# B&R Automation Studio project PLC code - cp (part 8)

#### Status.st
```iecst
ACTION Status:

	CASE Primer.Status.DeviceStatus OF
		PRIMER_TURNED_OFF:
			IF Primer.Inputs.xPrimerPresent THEN
				Primer.Status.DeviceStatus:=PRIMER_INIT;
			END_IF

		PRIMER_INIT:
			IF NOT Primer.Inputs.xPrimerPresent THEN
				Primer.Status.DeviceStatus:=PRIMER_TURNED_OFF;
			ELSIF Primer.Outputs.Physical.xPrepareToPrime OR Primer.Outputs.Physical.xRunTransport THEN
				Primer.Status.DeviceStatus:=PRIMER_PREPARING;
			END_IF

		PRIMER_PREPARING:
			IF Primer.Inputs.xTransportMoving THEN
				Primer.Status.DeviceStatus:=PRIMER_BELT_RUNNING;
			ELSIF NOT Primer.Outputs.Physical.xPrepareToPrime AND NOT Primer.Outputs.Physical.xRunTransport THEN
				Primer.Status.DeviceStatus:=PRIMER_INIT;
			END_IF

		PRIMER_BELT_RUNNING:
			IF NOT Primer.Inputs.xTransportMoving THEN
				Primer.Status.DeviceStatus:=PRIMER_INIT;
			END_IF
			IF Primer.Inputs.xReadyToPrime THEN
				Primer.Status.DeviceStatus:=PRIMER_READY;
			END_IF

		PRIMER_READY:
			IF NOT Primer.Inputs.xReadyToPrime THEN
				Primer.Status.DeviceStatus:=PRIMER_BELT_RUNNING;
			END_IF
			IF Primer.Inputs.xCoating THEN
				Primer.Status.DeviceStatus:=PRIMER_PRIMING;
			END_IF

		PRIMER_PRIMING:
			IF NOT Primer.Inputs.xCoating THEN
				Primer.Status.DeviceStatus:=PRIMER_READY;
			END_IF
			IF Primer.Inputs.xDryerInRun THEN
				Primer.Status.DeviceStatus:=PRIMER_DRYING;
			END_IF

		PRIMER_DRYING:
			IF NOT Primer.Inputs.xDryerInRun THEN
				Primer.Status.DeviceStatus:=PRIMER_PRIMING;
			END_IF

		PRIMER_FAULTED:
			IF NOT Primer.Inputs.xError THEN
				Primer.Status.DeviceStatus:=PRIMER_TURNED_OFF;
			END_IF

	END_CASE

	IF NOT Primer.Inputs.xPrimerPresent THEN
		Primer.Status.DeviceStatus:=PRIMER_TURNED_OFF;
	END_IF
	IF Primer.Status.DeviceStatus <> PRIMER_TURNED_OFF AND Primer.Inputs.xError THEN
		Primer.Status.DeviceStatus:=PRIMER_FAULTED;
	END_IF

	UpdateStatus;

	//Empty belt status
	tiTimeToEmpty := REAL_TO_TIME(60 * (Primer.Parameters.Hw.rPrimerLength + Primer.Parameters.rMediaLength) / Primer.Parameters.rSpeedSetPoint);
	tonEmptyBelt.IN := Primer.Inputs.xTransportMoving;
	tonEmptyBelt.PT := tiTimeToEmpty;
	tonEmptyBelt();
	IF Primer.Status.Comms.xModuleOk THEN
		Primer.Status.xBeltEmpty := Primer.Inputs.Comms.xBeltEmpty AND (tonEmptyBelt.Q OR NOT Primer.Inputs.xTransportMoving);
	ELSE
		Primer.Status.xBeltEmpty := (tonEmptyBelt.Q OR NOT Primer.Inputs.xTransportMoving);
	END_IF

END_ACTION

ACTION UpdateStatus:

	Primer.Status.Device.xTurnedOff 	:=	Primer.Status.DeviceStatus=PRIMER_TURNED_OFF;
	Primer.Status.Device.xInit			:=	Primer.Status.DeviceStatus=PRIMER_INIT;
	Primer.Status.Device.xPreparing 	:=	Primer.Status.DeviceStatus=PRIMER_PREPARING;
	Primer.Status.Device.xReady			:=	Primer.Status.DeviceStatus=PRIMER_READY;
	Primer.Status.Device.xPriming 		:=	Primer.Status.DeviceStatus=PRIMER_PRIMING;
	Primer.Status.Device.xFaulted 		:=	Primer.Status.DeviceStatus=PRIMER_FAULTED;

END_ACTION
```

### PrimerSim.typ
```iecst
TYPE
	PrimerSimCommands_typ : 	STRUCT
		CreateError : BOOL;
	END_STRUCT;
	PrimerSim_typ : 	STRUCT
		Commands : PrimerSimCommands_typ;
	END_STRUCT;
END_TYPE
```

### Program Logical/ExtPack/_Ancillaries/PrimerCtrl/PrimerSim/PrimerSim_v1/PrimerSim (IEC)

#### PrimerSim.st - Init, cyclic, exit code
```iecst
PROGRAM _INIT

	Primer ACCESS ADR(gPrimer);
	SimPrimer ACCESS ADR(gSimPrimer);

	Primer.Status.Comms.xModuleOk := TRUE;

END_PROGRAM

PROGRAM _CYCLIC
	(* Insert code here *)
	Primer ACCESS ADR(gPrimer);
	SimPrimer ACCESS ADR(gSimPrimer);

	IF NOT Primer.Parameters.xInstalled THEN
		Primer.Inputs := PrimerInputsReseted;
		RETURN;
	END_IF

	Primer.Inputs.xPrimerPresent:=TRUE;
	Primer.Inputs.Comms.xRemote := TRUE;
	Primer.Inputs.xError:=SimPrimer.Commands.CreateError;

	tonTransport.IN:= Primer.Outputs.Physical.xRunTransport;
	tonTransport.PT:= T#1s;
	tonTransport();
	Primer.Inputs.xTransportMoving:=tonTransport.Q;

	tonReady.IN:= Primer.Inputs.xTransportMoving AND Primer.Outputs.Physical.xPrepareToPrime;
	tonReady.PT:= T#2s;
	tonReady();
	Primer.Inputs.xReadyToPrime:=tonReady.Q;

	tonPrime.IN:= Primer.Inputs.xReadyToPrime AND Primer.Outputs.Physical.xRunPriming;
	tonPrime.PT:= T#1s;
	tonPrime();
	Primer.Inputs.xCoating:=tonPrime.Q;

	tonDry.IN:= Primer.Inputs.xCoating AND Primer.Outputs.Physical.xRunDryer;
	tonDry.PT:= T#1s;
	tonDry();
	Primer.Inputs.xDryerInRun:=tonDry.Q;

	Primer.Inputs.Comms.xBeltEmpty:=TRUE;
	Primer.Inputs.Comms.xCommsOK:=TRUE;

END_PROGRAM
```

#### PrimerSim.var - Local variables
```iecst
VAR
	SimPrimer : REFERENCE TO PrimerSim_typ;
	Primer : REFERENCE TO Primer_typ;
	tonTransport : TON;
	tonReady : TON;
	tonPrime : TON;
	tonBeltEmpty : TON;
	tonDry : TON;
	PrimerInputsReseted : {REDUND_UNREPLICABLE} PrimerInputs_typ;
END_VAR
```

- Dryer.graphml (not shown)

### Program Logical/ExtPack/_Ancillaries/DryerCtrl/DryerCtrl_v1/DryerCtrl (IEC)

#### Status.st
```iecst
ACTION Status:

	CASE Dryer.Status.DeviceStatus OF
		DRYER_TURNED_OFF:
			IF Dryer.Inputs.xInRemote THEN
				Dryer.Status.DeviceStatus:=DRYER_INIT;
			END_IF

		DRYER_INIT:
			IF Dryer.Outputs.xRunTransport OR Dryer.Outputs.xPrepareToDry THEN
				Dryer.Status.DeviceStatus:=DRYER_PREPARING;
			END_IF

		DRYER_PREPARING:
			IF Dryer.Inputs.xTransportMoving THEN
				Dryer.Status.DeviceStatus:=DRYER_BELTRUNNING;
			ELSIF NOT Dryer.Outputs.xRunTransport AND NOT Dryer.Outputs.xPrepareToDry THEN
				Dryer.Status.DeviceStatus:=DRYER_INIT;
			END_IF

		DRYER_BELTRUNNING:
			IF Dryer.Inputs.xReadyToDry THEN
				Dryer.Status.DeviceStatus:=DRYER_READY;
			ELSIF NOT Dryer.Inputs.xTransportMoving THEN
				Dryer.Status.DeviceStatus:=DRYER_INIT;
			END_IF

		DRYER_READY:
			IF Dryer.Inputs.xDrying THEN
				Dryer.Status.DeviceStatus:=DRYER_DRYING;
			ELSIF NOT Dryer.Inputs.xReadyToDry THEN
				Dryer.Status.DeviceStatus:=DRYER_INIT;
			END_IF

		DRYER_DRYING:
			IF NOT Dryer.Inputs.xDrying THEN
				Dryer.Status.DeviceStatus:=DRYER_INIT;
			END_IF

		DRYER_FAULTED:
			IF NOT Dryer.Inputs.xError THEN
				Dryer.Status.DeviceStatus:=DRYER_INIT;
			END_IF

	END_CASE

	IF NOT Dryer.Inputs.xCommsOK THEN
		Dryer.Status.DeviceStatus:=DRYER_TURNED_OFF;
	END_IF
	IF Dryer.Status.DeviceStatus <> DRYER_TURNED_OFF AND Dryer.Inputs.xError THEN
		Dryer.Status.DeviceStatus:=DRYER_FAULTED;
	END_IF

	UpdateStatus;

	//Empty belt status
	tiTimeToEmpty := REAL_TO_TIME(60 * (Dryer.Parameters.Hw.rDryerLength + Dryer.Parameters.rMediaLength) / Dryer.Parameters.rSpeedSetPoint);
	tonEmptyBelt.IN := Dryer.Inputs.xTransportMoving;
	tonEmptyBelt.PT := tiTimeToEmpty;
	tonEmptyBelt();
	IF Dryer.Inputs.xCommsOK THEN
		Dryer.Status.xBeltEmpty := Dryer.Inputs.xBeltEmpty AND (tonEmptyBelt.Q OR NOT Dryer.Inputs.xTransportMoving);
	ELSE
		Dryer.Status.xBeltEmpty := (tonEmptyBelt.Q OR NOT Dryer.Inputs.xTransportMoving);
	END_IF

END_ACTION

ACTION UpdateStatus:

	Dryer.Status.Device.xTurnedOff 		:=	Dryer.Status.DeviceStatus=DRYER_TURNED_OFF;
	Dryer.Status.Device.xInit 			:=	Dryer.Status.DeviceStatus=DRYER_INIT;
	Dryer.Status.Device.xPreparing 		:=	Dryer.Status.DeviceStatus=DRYER_PREPARING;
	Dryer.Status.Device.xBeltRunning 	:=	Dryer.Status.DeviceStatus=DRYER_BELTRUNNING;
	Dryer.Status.Device.xReadyToDry 	:=	Dryer.Status.DeviceStatus=DRYER_READY;
	Dryer.Status.Device.xDrying 		:=	Dryer.Status.DeviceStatus=DRYER_DRYING;
	Dryer.Status.Device.xFaulted 		:=	Dryer.Status.DeviceStatus=DRYER_FAULTED;

END_ACTION
```

#### Alarms.st
```iecst
ACTION Alarms:

	Dryer.Alarms.xNoDryerPresent:= NOT Dryer.Inputs.xInRemote;

	//IF NO Dryer, define that alarm and exit
	IF Dryer.Alarms.xNoDryerPresent THEN
		ResetAlarms;
		Dryer.Alarms.xNoDryerPresent:=TRUE;
	END_IF

	//Error
	IF Dryer.Inputs.xError THEN
		Dryer.Alarms.xError := TRUE;
	END_IF

	//Remote
	IF (NOT Dryer.Inputs.xInRemote) AND Dryer.Parameters.xLineInAuto THEN
		Dryer.Alarms.xNotRemote := TRUE;
	END_IF

	//Stop request
	IF (Dryer.Inputs.xStopButtonPressed) THEN
		Dryer.Alarms.xStopRequest := TRUE;
	END_IF

	//Summary
	Dryer.Alarms.xCriticalAlarm:= 	Dryer.Alarms.xError OR
									Dryer.Alarms.xNotRemote OR
									Dryer.Alarms.xStopRequest;

END_ACTION

ACTION ResetAlarms:
	Dryer.Alarms := AlarmsReseted;
END_ACTION
```

### Program Logical/ExtPack/_Ancillaries/OpvCtrl/OpvCtrl_v1/OpvCtrl (IEC)

#### Opv.st - Init, cyclic, exit code
```iecst
PROGRAM _CYCLIC

	OverVarnish ACCESS ADR(gOverVarnish);

	//Version
	OverVarnish.Status.Version.iVersion0 := OverVarnish.Inputs.Comms.iVersion1;
	OverVarnish.Status.Version.iVersion1 := OverVarnish.Inputs.Comms.iVersion2;
	OverVarnish.Status.Version.iVersion2 := OverVarnish.Inputs.Comms.iVersion3;
	OverVarnish.Status.Version.iVersion3 := OverVarnish.Inputs.Comms.iVersion4;

	//Model evaluation
	iOpvModel.0 := OverVarnish.Inputs.xModelInput[0];
	iOpvModel.1 := OverVarnish.Inputs.xModelInput[1];
	iOpvModel.2 := OverVarnish.Inputs.xModelInput[2];

	OverVarnish.Parameters.xInstalled := iOpvModel>0;

	//Specify Type of Opv Model
	OverVarnish.Status.iModel := iOpvModel;
	CASE iOpvModel OF
		1: OverVarnish.Status.OpvType := OPVTY_GIARDINA;
		2: OverVarnish.Status.OpvType := OPVTY_DMS;
		3: OverVarnish.Status.OpvType := OPVTY_TECLIGHTING;
		ELSE OverVarnish.Status.OpvType := OPVTY_UNDEFINED;
	END_CASE

	IF NOT OverVarnish.Parameters.xInstalled OR NOT OverVarnish.ParSw.xEnabled THEN
		ResetAlarms;
		OverVarnish.Outputs := OutputsReset;
		OverVarnish.Commands:=ResetCommands;
		OverVarnish.Status.DeviceStatus:=OPV_TURNED_OFF;
		CopyOfWriteData := EraseWriteData;
		UpdateStatus;
		RETURN;
	END_IF

	IF OverVarnish.Commands.xResetAlarms THEN ResetAlarms; END_IF

	Configuration;

	IF NOT OverVarnish.Parameters.xSimulationMode THEN
		AssignDataComms;
	END_IF

	Status;

	//Erasing data when ancillary not in remote
	IF NOT OverVarnish.Inputs.Comms.xRemote THEN
		CopyOfWriteData := EraseWriteData;
	END_IF

	Alarms;

	IF OverVarnish.Status.Device.xFaulted OR OverVarnish.Status.Device.xTurnedOff OR NOT OverVarnish.Parameters.xLineInAuto THEN
		OverVarnish.Status.CtrlStatus:=OPVCTRL_STOPPED;
	END_IF

	CASE OverVarnish.Status.CtrlStatus OF
		OPVCTRL_STOPPED:
			//Actions
			OverVarnish.Outputs.Physical := PhysicalOutputsReset;

			//Transition
			IF OverVarnish.Commands.xPrepare THEN
				xEnablePriming:= OverVarnish.ParSw.xEnablePriming AND OverVarnish.Orders.xEnablePriming;
				OverVarnish.Status.CtrlStatus:=OPVCTRL_PREPARING;
			END_IF

		OPVCTRL_STOPPING:
			//Actions
			OverVarnish.Outputs.Physical := PhysicalOutputsReset;

			//Transition
			IF OverVarnish.Status.DeviceStatus=OPV_TURNED_OFF OR OverVarnish.Status.DeviceStatus=OPV_INIT THEN
				OverVarnish.Status.CtrlStatus:=OPVCTRL_STOPPED;
			END_IF

		OPVCTRL_CONTROLSTOPPING:
			//Wait to have the belt empty and send the Stop order
			IF OverVarnish.Status.xBeltEmpty AND EDGEPOS(OverVarnish.Orders.xDisableReadBlock) OR NOT OverVarnish.Inputs.xTransportMoving THEN
				OverVarnish.Status.CtrlStatus:=OPVCTRL_STOPPING;
			END_IF

		OPVCTRL_PREPARING:
			//Actions

			IF xEnablePriming THEN
				OverVarnish.Outputs.Physical.xRunTransport:=TRUE;
				OverVarnish.Outputs.Physical.xPrepareToPrime:=TRUE;
				//Transition
				IF OverVarnish.Status.DeviceStatus=OPV_READY THEN
					OverVarnish.Status.CtrlStatus:=OPVCTRL_PREPARED;
				END_IF

			ELSE
				OverVarnish.Outputs.Physical.xRunTransport:=TRUE;
				//Transition
				IF OverVarnish.Status.DeviceStatus=OPV_BELT_RUNNING THEN
					OverVarnish.Status.CtrlStatus:=OPVCTRL_PREPARED;
				END_IF

			END_IF

		OPVCTRL_PAUSED,
		OPVCTRL_PREPARED:
			//Actions
			IF OverVarnish.Commands.xStart THEN
				OverVarnish.Status.CtrlStatus:=OPVCTRL_STARTING;
			END_IF

		OPVCTRL_STARTING:
			//Actions
			IF xEnablePriming THEN
				OverVarnish.Outputs.Physical.xRunPriming:=TRUE;
				IF OverVarnish.Status.DeviceStatus=OPV_PRIMING THEN
					OverVarnish.Outputs.Physical.xRunDryer:=TRUE;
				END_IF
				//Transition
				IF OverVarnish.Status.DeviceStatus=OPV_DRYING THEN
					OverVarnish.Status.CtrlStatus:=OPVCTRL_WORKING;
				END_IF

			ELSE
				OverVarnish.Outputs.Physical.xRunTransport:=TRUE;
				IF OverVarnish.Status.DeviceStatus=OPV_BELT_RUNNING THEN
					OverVarnish.Status.CtrlStatus:=OPVCTRL_WORKING;
				END_IF

			END_IF

			//Transition
			IF OverVarnish.Commands.xPause THEN
				OverVarnish.Status.CtrlStatus:=OPVCTRL_PAUSING;
			END_IF

		OPVCTRL_WORKING:
			IF OverVarnish.Commands.xPause THEN
				OverVarnish.Status.CtrlStatus:=OPVCTRL_PAUSING;
			END_IF

		OPVCTRL_PAUSING:
			//Wait to empty the Belt to avoid media inside
			IF OverVarnish.Status.xBeltEmpty THEN
				IF xEnablePriming THEN
					OverVarnish.Outputs.Physical.xRunDryer:=FALSE;
					//Transition
					IF OverVarnish.Status.DeviceStatus=OPV_PRIMING THEN
						OverVarnish.Status.CtrlStatus:=OPVCTRL_PAUSED;
					END_IF

				ELSE
					IF OverVarnish.Status.DeviceStatus=OPV_INIT OR OverVarnish.Status.DeviceStatus=OPV_BELT_RUNNING THEN
						OverVarnish.Status.CtrlStatus:=OPVCTRL_PAUSED;
					END_IF
				END_IF
			END_IF

	END_CASE

	IF OverVarnish.Commands.xStop THEN
		OverVarnish.Status.CtrlStatus:=OPVCTRL_STOPPING;
	ELSIF OverVarnish.Commands.xControlStop THEN
		OverVarnish.Status.CtrlStatus:=OPVCTRL_CONTROLSTOPPING;
	END_IF

	//Store the history of the status to easy the debug
	IF OverVarnish.Status.CtrlStatus<>StateHistory[0] THEN
		FOR iIndexHistory:=iHistoryLines TO 1 BY -1 DO
			StateHistory[iIndexHistory]:=StateHistory[iIndexHistory-1];
		END_FOR;
		StateHistory[0]:=OverVarnish.Status.CtrlStatus;
	END_IF

	//Fall down the commands
	OverVarnish.Commands:=ResetCommands;

END_PROGRAM
```

#### AssignDataComms.st
```iecst
ACTION AssignDataComms:

	//Active modbus slave diagnosis when ancillary is enabled. This parameter must remain to TRUE from then on.
	//Just would be set to FALSE via UaExpert, to reset historic errors when ancillary is disabled
	OverVarnish.Parameters.xActiveSlaveDiagnosis := TRUE;

	xBoardParametersChanged := 	(OverVarnish.Parameters.Media.rWidth<>rPrevWidth) OR
								(OverVarnish.Parameters.Media.rLength<>rPrevLength) OR
								(OverVarnish.Parameters.Media.rThickness<>rPrevThickness) OR
								(OverVarnish.Parameters.Media.rGap<>rPrevGap);

	rPrevWidth:=OverVarnish.Parameters.Media.rWidth;
	rPrevLength:=OverVarnish.Parameters.Media.rLength;
	rPrevThickness:=OverVarnish.Parameters.Media.rThickness;
	rPrevGap:=OverVarnish.Parameters.Media.rGap;

	tof_BoardParametersChanged.IN:=xBoardParametersChanged;
	tof_BoardParametersChanged.PT:=t#1s;
	tof_BoardParametersChanged();

	IF OverVarnish.Status.OpvType = OPVTY_DMS THEN
		DmsComms;
	ELSE
		DefaultPrimerComms;
	END_IF

	//Disabling writting after some time active. To test
	tonDisableWrittingOfData.IN:= NOT xDisableWriteData;
	tonDisableWrittingOfData.PT:= T#1000ms;
	tonDisableWrittingOfData();

	IF tonDisableWrittingOfData.Q THEN
		xDisableWriteData := TRUE;
	END_IF

	FOR iIndex:=1 TO 25 DO
		IF gToWriteDataModbOpv[iIndex]<>CopyOfWriteData[iIndex] THEN
			xDisableWriteData := FALSE;
		END_IF
	END_FOR

	OverVarnish.Orders.xDisableWriteBlock := xDisableWriteData;

	//Copying previous data
	CopyOfWriteData := gToWriteDataModbOpv;

END_ACTION

ACTION DmsComms:

			/////////////////
			//Pre bits treatment
			OverVarnish.Outputs.Comms.iControl.1 := OverVarnish.Commands.xEnteringMedia;
			OverVarnish.Outputs.Comms.iControl.2 := OverVarnish.Commands.xNewBoardParameters:=tof_BoardParametersChanged.Q;
			//OverVarnish.Outputs.Comms.iControl.3 := ;
			OverVarnish.Outputs.Comms.iControl.4 := TRUE; //OverVarnish.Outputs.Comms.xLineAirSupply;
			OverVarnish.Outputs.Comms.iControl.5 := OverVarnish.Parameters.LineState = LINE_PREPARING_EMPTYBELT OR
													OverVarnish.Parameters.LineState = LINE_STARTING_EMPTYBELT OR
													OverVarnish.Parameters.LineState = LINE_BELT_EMPTYING;

			OverVarnish.Outputs.Comms.iControl2.13 := FALSE; //Single line:0, Double line: 1
			OverVarnish.Outputs.Comms.iControl2.15 := TRUE; //Edge:0, Center: 1

			//Write Registers
			gToWriteDataModbOpv[1] := REAL_TO_UINT(OverVarnish.Parameters.Media.rWidth*10);
			gToWriteDataModbOpv[2] := REAL_TO_UINT(OverVarnish.Parameters.Media.rLength*10);
			gToWriteDataModbOpv[3] := REAL_TO_UINT(OverVarnish.Parameters.Media.rThickness*10);
			gToWriteDataModbOpv[4] := REAL_TO_UINT(OverVarnish.Parameters.Media.rGap*10);
			//gToWriteDataModbOpv[5] := ;
			gToWriteDataModbPrimer[6] := REAL_TO_UINT(OverVarnish.Parameters.rLineAccelRate*60); //150;
			gToWriteDataModbPrimer[7] := REAL_TO_UINT(OverVarnish.Parameters.rLineDecelRate*60); //150;
			gToWriteDataModbOpv[8] := REAL_TO_UINT(OverVarnish.Parameters.rSpeedSetPoint*100);
			gToWriteDataModbOpv[9] := OverVarnish.Outputs.Comms.iControl;
			gToWriteDataModbOpv[10] := OverVarnish.Outputs.Comms.iControl2;
			//gToWriteDataModbOpv[11] := ;
			//gToWriteDataModbOpv[12] := ;
			//gToWriteDataModbOpv[13] := ;
			gToWriteDataModbOpv[14] := REAL_TO_UINT(OverVarnish.Parameters.rLineAccelRate*60); //150;
			gToWriteDataModbOpv[15] := REAL_TO_UINT(OverVarnish.Parameters.rLineDecelRate*60); //150;
			(*
			gToWriteDataModbOpv[16] := ;
			gToWriteDataModbOpv[17] := ;
			gToWriteDataModbOpv[18] := ;
			gToWriteDataModbOpv[19] := ;
			gToWriteDataModbOpv[20] := ;
			gToWriteDataModbOpv[21] := ;
			gToWriteDataModbOpv[22] := ;
			gToWriteDataModbOpv[23] := ;
			gToWriteDataModbOpv[24] := ;
			gToWriteDataModbOpv[25] := ;
			*)

		////////////////
		//Read Registers
		IF OverVarnish.Status.Comms.xModuleOk THEN
			OverVarnish.Inputs.Comms.iStatus := gReceivedDataModbOpv[1];
			//OverVarnish.Inputs.Comms. := gReceivedDataModbOpv[2];
			OverVarnish.Inputs.Comms.uiCoaterRollerSpeed := gReceivedDataModbOpv[3];
			OverVarnish.Inputs.Comms.uiTransportSpeed := gReceivedDataModbOpv[4];
			(*
			:= gReceivedDataModbOpv[5];
			:= gReceivedDataModbOpv[6];
			:= gReceivedDataModbOpv[7];
			:= gReceivedDataModbOpv[8];
			:= gReceivedDataModbOpv[9];
			:= gReceivedDataModbOpv[10];
			:= gReceivedDataModbOpv[11];
			:= gReceivedDataModbOpv[12];
			:= gReceivedDataModbOpv[13];
			:= gReceivedDataModbOpv[14];
			:= gReceivedDataModbOpv[15];
			*)
			OverVarnish.Inputs.Comms.iVersion1 := gReceivedDataModbOpv[16];
			OverVarnish.Inputs.Comms.iVersion2 := gReceivedDataModbOpv[17];
			OverVarnish.Inputs.Comms.iVersion3 := gReceivedDataModbOpv[18];
			OverVarnish.Inputs.Comms.iVersion4 := gReceivedDataModbOpv[19];
			(*
			:= gReceivedDataModbOpv[20];
			:= gReceivedDataModbOpv[21];
			:= gReceivedDataModbOpv[22];
			:= gReceivedDataModbOpv[23];
			:= gReceivedDataModbOpv[24];
			:= gReceivedDataModbOpv[25];
			*)

	END_IF

		//Post bit treatment
		OverVarnish.Inputs.Comms.xRemote := OverVarnish.Inputs.Comms.iStatus.1;
		OverVarnish.Inputs.Comms.xBeltEmpty := OverVarnish.Inputs.Comms.iStatus.3;
		OverVarnish.Inputs.Comms.xStopButtonPressed := OverVarnish.Inputs.Comms.iStatus.10;

END_ACTION

ACTION DefaultPrimerComms:

		/////////////////
		//Pre bits treatment
		//OverVarnish.Outputs.Comms.iControl.0 := ;
		//OverVarnish.Outputs.Comms.iControl.1 := ;
		OverVarnish.Outputs.Comms.iControl.2 := OverVarnish.Commands.xNewBoardParameters := tof_BoardParametersChanged.Q;
		//Primer.Outputs.Comms.iControl.3 := ;
		//Primer.Outputs.Comms.iControl.4 := ;
		OverVarnish.Outputs.Comms.iControl.5 := OverVarnish.Parameters.LineState = LINE_PREPARING_EMPTYBELT OR
												OverVarnish.Parameters.LineState = LINE_STARTING_EMPTYBELT OR
												OverVarnish.Parameters.LineState = LINE_BELT_EMPTYING;

		//Write Registers
		gToWriteDataModbOpv[1] := OverVarnish.Outputs.Comms.iControl;
		gToWriteDataModbOpv[2] := REAL_TO_UINT(OverVarnish.Parameters.Media.rLength*10);
		gToWriteDataModbOpv[3] := REAL_TO_UINT(OverVarnish.Parameters.Media.rWidth*10);
		gToWriteDataModbOpv[4] := REAL_TO_UINT(OverVarnish.Parameters.Media.rThickness*10);
		gToWriteDataModbOpv[5] := REAL_TO_UINT(OverVarnish.Parameters.Media.rGap*10);
		gToWriteDataModbPrimer[6] := REAL_TO_UINT(OverVarnish.Parameters.rLineAccelRate*60); //150;
		gToWriteDataModbPrimer[7] := REAL_TO_UINT(OverVarnish.Parameters.rLineDecelRate*60); //150;
		gToWriteDataModbOpv[8] := REAL_TO_UINT(OverVarnish.Parameters.rSpeedSetPoint*10);
		(*
		gToWriteDataModbOpv[9] := ;
		gToWriteDataModbOpv[10] := ;
		gToWriteDataModbOpv[11] := ;

		gToWriteDataModbOpv[12] := ;
		gToWriteDataModbOpv[13] := ;
		gToWriteDataModbOpv[14] := ;
		gToWriteDataModbOpv[15] := ;
		gToWriteDataModbOpv[16] := ;
		gToWriteDataModbOpv[17] := ;
		gToWriteDataModbOpv[18] := ;
		gToWriteDataModbOpv[19] := ;
		gToWriteDataModbOpv[20] := ;
		gToWriteDataModbOpv[21] := ;
		gToWriteDataModbOpv[22] := ;
		gToWriteDataModbOpv[23] := ;
		gToWriteDataModbOpv[24] := ;
		gToWriteDataModbOpv[25] := ;
		*)

		////////////////
		//Read Registers
		IF OverVarnish.Status.Comms.xModuleOk THEN
			OverVarnish.Inputs.Comms.iStatus := gReceivedDataModbOpv[1];
			//Primer.Inputs.Comms. := gReceivedDataModbOpv[2];
			OverVarnish.Inputs.Comms.uiCoaterRollerSpeed := gReceivedDataModbOpv[3];
			OverVarnish.Inputs.Comms.uiTransportSpeed := gReceivedDataModbOpv[4];
			(*
			:= gReceivedDataModbOpv[5];
			:= gReceivedDataModbOpv[6];
			:= gReceivedDataModbOpv[7];
			:= gReceivedDataModbOpv[8];
			:= gReceivedDataModbOpv[9];
			:= gReceivedDataModbOpv[10];
			:= gReceivedDataModbOpv[11];
			:= gReceivedDataModbOpv[12];
			:= gReceivedDataModbOpv[13];
			:= gReceivedDataModbOpv[14];
			:= gReceivedDataModbOpv[15];
			*)
			OverVarnish.Inputs.Comms.iVersion1 := gReceivedDataModbOpv[16];
			OverVarnish.Inputs.Comms.iVersion2 := gReceivedDataModbOpv[17];
			OverVarnish.Inputs.Comms.iVersion3 := gReceivedDataModbOpv[18];
			OverVarnish.Inputs.Comms.iVersion4 := gReceivedDataModbOpv[19];
			(*
			:= gReceivedDataModbOpv[20];
			:= gReceivedDataModbOpv[21];
			:= gReceivedDataModbOpv[22];
			:= gReceivedDataModbOpv[23];
			:= gReceivedDataModbOpv[24];
			:= gReceivedDataModbOpv[25];
			*)
		END_IF

		//Post bit treatment
		// := OverVarnish.Inputs.Comms.iStatus.0;
		// := OverVarnish.Inputs.Comms.iStatus.1;
		// := OverVarnish.Inputs.Comms.iStatus.2;
		// := OverVarnish.Inputs.Comms.iStatus.3;
		// := OverVarnish.Inputs.Comms.iStatus.4;
		// := OverVarnish.Inputs.Comms.iStatus.5;
		// := OverVarnish.Inputs.Comms.iStatus.6;
		// := OverVarnish.Inputs.Comms.iStatus.7;
		OverVarnish.Inputs.Comms.xRemote := OverVarnish.Inputs.Comms.iStatus.8;
		OverVarnish.Inputs.Comms.xBeltEmpty := OverVarnish.Inputs.Comms.iStatus.9;
		// := OverVarnish.Inputs.Comms.iStatus.10;

END_ACTION
```

### Opv.typ
```iecst
TYPE
	OPVCtrlStatus_enum :
		(
		OPVCTRL_STOPPED,
		OPVCTRL_STOPPING,
		OPVCTRL_PREPARING,
		OPVCTRL_PREPARED,
		OPVCTRL_PAUSING,
		OPVCTRL_PAUSED,
		OPVCTRL_STARTING,
		OPVCTRL_WORKING,
		OPVCTRL_CONTROLSTOPPING
		);
	OPVStatus_enum :
		(
		OPV_TURNED_OFF,
		OPV_INIT,
		OPV_PREPARING,
		OPV_READY,
		OPV_DRYING,
		OPV_FAULTED,
		OPV_PRIMING,
		OPV_BELT_RUNNING
		);
	OpvType_enum :
		(
		OPVTY_UNDEFINED,
		OPVTY_GIARDINA,
		OPVTY_DMS,
		OPVTY_TECLIGHTING
		);
	OPVCommsInputs_typ : 	STRUCT
		xCommsOK : BOOL; (*Modbus communications are working properly*)
		uiTransportSpeed : UINT;
		uiCoaterRollerSpeed : UINT;
		xRemote : BOOL;
		xBeltEmpty : BOOL; (*Belt empty in the device*)
		iVersion1 : INT; (*Machine platform (Nozomi = 1)*)
		iVersion2 : INT; (*Machine project (C18000 = 0 / C14000 = 1)*)
		iVersion3 : INT; (*Hardware version*)
		iVersion4 : INT; (*Sotfware version*)
		iStatus : INT; (*Status word*)
		xStopButtonPressed : BOOL;
	END_STRUCT;
	OPVInputs_typ : 	STRUCT
		xOPVPresent : BOOL;
		xReadyToPrime : BOOL;
		xCoating : BOOL;
		xError : BOOL;
		xCoatingLevelLow : BOOL;
		xTransportMoving : BOOL;
		xDryerInRun : BOOL;
		xCriticalAlarm : BOOL;
		iCoaterModel : INT;
		xModelInput : ARRAY[0..2]OF BOOL;
		xNoPowered : BOOL;
		Comms : OPVCommsInputs_typ;
	END_STRUCT;
	OPVOutputs_typ : 	STRUCT
		Physical : OPVPhysicalOutputs_typ;
		Comms : OPVCommsOutputs_typ;
	END_STRUCT;
	OPVAlarms_typ : 	STRUCT
		xError : BOOL;
		xNoOPVPresent : BOOL;
		xCoatingLevelLow : BOOL;
		xAnyAlarm : BOOL;
		xNotRemote : BOOL;
		xCoatingRecircNotEnabled : BOOL;
		xNoPowered : BOOL;
		xCriticalAlarm : BOOL;
		xWarningAlarm : BOOL;
		xCommsError : BOOL;
		xStopRequest : BOOL; (*Stop request from Dryer when physical stop button is pressed*)
	END_STRUCT;
	OPVParametersSw_typ : 	STRUCT
		xEnabled : BOOL; (*This variable replaces the previous "xThereIs". Activated by SW*)
		xEnablePriming : BOOL; (*Priming enabled from SW*)
	END_STRUCT;
	OPVParametersHw_typ : 	STRUCT
		iMaxMediaWidth : UINT; (*Maximum media width allowed in mm*)
		iMinMediaWidth : UINT; (*Minimum media width allowed in mm*)
		iMaxMediaLength : UINT; (*Maximum media length allowed in mm*)
		iMinMediaLength : UINT; (*Minimum media length allowed in mm*)
		rOPVLength : REAL; (*Length in mm*)
		rMaxSpeed : REAL := 100.0; (*Maximum speed allowed in m/min*)
		iMinMediaThickness : UINT; (*Minimum media height allowed in tenth of mm*)
		iMaxMediaThickness : UINT; (*Maximum media height allowed in tenth of mm*)
		xDoubleLineAllowed : BOOL; (*Active when allows double line printing*)
	END_STRUCT;
	OPVParameters_typ : 	STRUCT
		xInstalled : BOOL;
		xSimulationMode : BOOL; (*Defined by the configuration in Automation Studio*)
		xAlrPresent : BOOL;
		xLineInAuto : BOOL;
		xPreviousDeviceStopped : BOOL; (*Length in mm*)
		rMediaLength : REAL; (*Length in mm*)
		Media : OPVMediaParameters;
		rLineAccelRate : REAL := 2; (*mm/s2 (2.5m/s2*60=150mpm/s)*)
		rLineDecelRate : REAL := 2; (*mm/s2 (2.5m/s2*60=150mpm/s)*)
		xDoubleLine : BOOL;
		LineState : LineStatus_enum;
		LineStatusSummary : LineControlStatusSummarized;
		Hw : OPVParametersHw_typ;
		xActiveSlaveDiagnosis : BOOL;
		rSpeedSetPoint : REAL;
	END_STRUCT;
	OPVCommands_typ : 	STRUCT
		xStart : BOOL; (*Edge commands. Reseted when managed*)
		xPrepare : BOOL; (*Edge commands. Reseted when managed*)
		xPause : BOOL; (*Edge commands. Reseted when managed*)
		xBelEmpty : BOOL; (*Edge commands. Reseted when managed*)
		xControlStop : BOOL; (*Edge commands. Reseted when managed*)
		xStop : BOOL; (*Edge commands. Reseted when managed*)
		xThereIsOPV : BOOL;
		xResetAlarms : BOOL;
		xEnteringMedia : BOOL;
		xNewBoardParameters : BOOL; (*Pulse to let know board paramters have changed*)
	END_STRUCT;
	OPVDeviceStatus_typ : 	STRUCT
		xTurnedOff : BOOL;
		xInit : BOOL;
		xPreparing : BOOL;
		xEmpty : BOOL;
		xReady : BOOL;
		xPriming : BOOL;
		xDrying : BOOL;
		xFaulted : BOOL;
	END_STRUCT;
	OPVStatus_typ : 	STRUCT
		iModel : USINT; (*Model of the Device. 0:Retroflex*)
		Version : EFI_version_typ;
		CtrlStatus : OPVCtrlStatus_enum;
		DeviceStatus : OPVStatus_enum;
		Device : OPVDeviceStatus_typ;
		xBeltEmpty : BOOL;
		OpvType : OpvType_enum;
		Comms : OPVCommsStatus_typ;
	END_STRUCT;
	Opv_typ : 	STRUCT
		Inputs : OPVInputs_typ;
		Outputs : OPVOutputs_typ;
		Alarms : OPVAlarms_typ;
		ParSw : OPVParametersSw_typ;
		Parameters : OPVParameters_typ;
		Commands : OPVCommands_typ;
		Status : OPVStatus_typ;
		Orders : OpvOrders_typ;
	END_STRUCT;
	OPVPhysicalOutputs_typ : 	STRUCT
		xPrepareToPrime : BOOL;
		xRunPriming : BOOL;
		xRunTransport : BOOL;
		xRunDryer : BOOL;
		xEnabledNormalDecel : BOOL;
	END_STRUCT;
	OPVCommsOutputs_typ : 	STRUCT
		iControl : INT; (*Status word*)
		iControl2 : INT; (*Status word*)
	END_STRUCT;
	OPVMediaParameters : 	STRUCT
		rThickness : REAL; (*Tile thickness to print from gui in mm*)
		rWidth : REAL; (*Board's width in mm*)
		rGap : REAL; (*Gap between boards in mm*)
		rLength : REAL; (*Board's length in mm*)
		rOffsetRegisterL1 : REAL; (*Board's width in mm*)
		rOffsetRegisterL2 : REAL; (*Board's width in mm*)
	END_STRUCT;
	OPVCommsStatus_typ : 	STRUCT
		xModuleOk : BOOL;
		ModSlaveState : UINT;
		LastError : UINT;
		LastErrorBlockNum : UINT;
		xStopButtonPressed : BOOL;
		ActOverloadError : BOOL;
		ActModbusError : BOOL;
		ActSlvConError : BOOL;
		ActRefreshError : BOOL;
		ActInternalError : BOOL;
		ActConfError : BOOL;
		HistOverloadError : BOOL;
		HistModbusError : BOOL;
		HistSlvConError : BOOL;
		HistRefreshError : BOOL;
		HistInternalError : BOOL;
		HistConfError : BOOL;
		ModbusErrorCnt : UINT;
		ModbusConErrorCnt : UINT;
		ModbusPktRefreshTimeoutCnt : UINT;
		ModbusPktPendPerSec : UINT;
		ModbusMeanResponseTime : UINT;
	END_STRUCT;
	OpvOrders_typ : 	STRUCT
		xDisableWriteBlock : BOOL;
		xDisableReadBlock : BOOL;
		xEnablePriming : BOOL; (*Priming enabled from printer/line*)
	END_STRUCT;
END_TYPE
```

### Program Logical/ExtPack/_Ancillaries/OpvCtrl/OpvSim/OpvSim_v1/OpvSim (IEC)

#### OpvSim.st - Init, cyclic, exit code
```iecst
PROGRAM _INIT

	Opv ACCESS ADR(gOverVarnish);

	Opv.Status.Comms.xModuleOk := TRUE;

END_PROGRAM

PROGRAM _CYCLIC
	(* Insert code here *)
	Opv ACCESS ADR(gOverVarnish);
	SimOpv ACCESS ADR(gSimOverVarnish);

	Opv.Inputs.xOPVPresent:=TRUE;
	Opv.Inputs.Comms.xRemote := TRUE;
	Opv.Inputs.xError:=SimOpv.Commands.CreateError;

	tonTransport.IN:= Opv.Outputs.Physical.xRunTransport;
	tonTransport.PT:= T#1s;
	tonTransport();
	Opv.Inputs.xTransportMoving:=tonTransport.Q;

	tonReady.IN:= Opv.Inputs.xTransportMoving AND Opv.Outputs.Physical.xPrepareToPrime;
	tonReady.PT:= T#2s;
	tonReady();
	Opv.Inputs.xReadyToPrime:=tonReady.Q;

	tonPrime.IN:= Opv.Inputs.xReadyToPrime AND Opv.Outputs.Physical.xRunPriming;
	tonPrime.PT:= T#1s;
	tonPrime();
	Opv.Inputs.xCoating:=tonPrime.Q;

	tonDry.IN:= Opv.Inputs.xCoating AND Opv.Outputs.Physical.xRunDryer;
	tonDry.PT:= T#1s;
	tonDry();
	Opv.Inputs.xDryerInRun:=tonDry.Q;

	Opv.Inputs.Comms.xBeltEmpty:=TRUE;
	Opv.Inputs.Comms.xCommsOK:=TRUE;

END_PROGRAM
```

### Program Logical/ExtPack/_Ancillaries/StackerCtrl/StackerCtrl_v1/StackerCtrl (IEC)

#### Stacker.st - Init, cyclic, exit code
```iecst
PROGRAM _CYCLIC

	Stacker ACCESS ADR(gStacker);

	//Version
	Stacker.Status.Version.iVersion0 := Stacker.Inputs.Comms.iVersion1;
	Stacker.Status.Version.iVersion1 := Stacker.Inputs.Comms.iVersion2;
	Stacker.Status.Version.iVersion2 := Stacker.Inputs.Comms.iVersion3;
	Stacker.Status.Version.iVersion3 := Stacker.Inputs.Comms.iVersion4;

	//Model evaluation
	iStackerModel.0 := Stacker.Inputs.xModelInput[0];
	iStackerModel.1 := Stacker.Inputs.xModelInput[1];
	iStackerModel.2 := Stacker.Inputs.xModelInput[2];

	Stacker.Parameters.xInstalled := iStackerModel>0;

	//Specify Type of Stacker Model
	Stacker.Status.iModel := iStackerModel;
	CASE iStackerModel OF
		1: Stacker.Status.StackerType := STACKERTY_FULL_S;
		2: Stacker.Status.StackerType := STACKERTY_BUNDLE_S;
		ELSE Stacker.Status.StackerType := STACKERTY_UNDEFINED;
	END_CASE

	IF NOT Stacker.Parameters.xInstalled OR NOT Stacker.ParSw.xEnabled THEN
		ResetAlarms;
		Stacker.Outputs := OutputsReset;
		Stacker.Commands:=ResetCommands;
		Stacker.Status.DeviceStatus:=STACKER_TURNED_OFF;
		CopyOfWriteData := EraseWriteData;
		UpdateStatus;
		RETURN;
	END_IF

	IF Stacker.Commands.xResetAlarms THEN ResetAlarms; END_IF

	Configuration;

	Status;

	IF NOT Stacker.Parameters.xSimulationMode THEN
		AssignDataComms;
	END_IF

	//Erasing data when ancillary not in remote
	IF NOT Stacker.Inputs.Comms.xRemote THEN
		CopyOfWriteData := EraseWriteData;
	END_IF

	Alarms;

	IF Stacker.Status.Device.xFaulted OR Stacker.Status.Device.xTurnedOff OR NOT Stacker.Parameters.xLineInAuto THEN
		Stacker.Status.CtrlStatus:=STACKERCTRL_STOPPED;
		Stacker.Outputs := OutputsReset; //To reset outputs in this conditions instead of when stacker is stopped. So outputs as ejectstack, stackeject
	END_IF

	ton_ControlStopping.IN := Stacker.Status.CtrlStatus = STACKERCTRL_CONTROLSTOPPING;
	ton_ControlStopping.PT := T#1s;
	ton_ControlStopping();

	CASE Stacker.Status.CtrlStatus OF
		STACKERCTRL_STOPPED:
			//Actions
			Stacker.Outputs := OutputsReset;

			IF Stacker.Status.DeviceStatus=STACKER_INIT AND Stacker.Commands.xPrepare THEN
				Stacker.Status.CtrlStatus:=STACKERCTRL_PREPARING;
			END_IF

		STACKERCTRL_STOPPING:
			//Actions
			Stacker.Outputs := OutputsReset;

			//Transition
			IF Stacker.Status.DeviceStatus=STACKER_TURNED_OFF OR Stacker.Status.DeviceStatus=STACKER_INIT THEN
				Stacker.Status.CtrlStatus:=STACKERCTRL_STOPPED;
			END_IF

		STACKERCTRL_CONTROLSTOPPING:
			//Wait to have the belt empty and send the Stop order
			tonEmptyBelt.IN := Stacker.Parameters.xPreviousDeviceStopped;
			IF (Stacker.Status.xBeltEmpty AND ton_ControlStopping.Q AND EDGEPOS(Stacker.Orders.xDisableReadBlock)) OR NOT Stacker.Inputs.xRunning THEN
				Stacker.Status.CtrlStatus:=STACKERCTRL_STOPPING;
			END_IF

		STACKERCTRL_PREPARING:
			Stacker.Outputs.xPrepareToStack:=TRUE;
			IF Stacker.Status.DeviceStatus=STACKER_READY THEN
				Stacker.Status.CtrlStatus:=STACKERCTRL_PREPARED;
			END_IF

		STACKERCTRL_PAUSED,
		STACKERCTRL_PREPARED:
			IF Stacker.Commands.xStart THEN
				Stacker.Status.CtrlStatus:=STACKERCTRL_STARTING;
			END_IF

		STACKERCTRL_STARTING:
			Stacker.Outputs.xRun:=TRUE;
			IF Stacker.Status.DeviceStatus=STACKER_WORKING THEN
				Stacker.Status.CtrlStatus:=STACKERCTRL_WORKING;
			END_IF

		STACKERCTRL_WORKING:
			Stacker.Outputs.xRejectSheet := Stacker.Orders.xRejectSheet;
			IF Stacker.Commands.xPause THEN
				Stacker.Status.CtrlStatus:=STACKERCTRL_PAUSING;
			END_IF

		STACKERCTRL_PAUSING:
			//Wait to empty the Belt to avoid media inside
			IF Stacker.Status.xBeltEmpty THEN
				Stacker.Status.CtrlStatus:=STACKERCTRL_PAUSED;
			END_IF

	END_CASE

	IF Stacker.Commands.xStop THEN
		Stacker.Status.CtrlStatus:=STACKERCTRL_STOPPING;
	ELSIF Stacker.Commands.xControlStop THEN
		Stacker.Status.CtrlStatus:=STACKERCTRL_CONTROLSTOPPING;
	END_IF

	//Store the history of the status to easy the debug
	IF Stacker.Status.CtrlStatus<>StateHistory[0] THEN
		FOR iIndexHistory:=iHistoryLines TO 1 BY -1 DO
			StateHistory[iIndexHistory]:=StateHistory[iIndexHistory-1];
		END_FOR;
		StateHistory[0]:=Stacker.Status.CtrlStatus;
	END_IF

	//Commands sent by SW
	tp_CleanBelts(IN:=Stacker.Commands.xCleanBelts, PT:=T#2S);
	tp_EjectPileStack(IN:=Stacker.Commands.xEjectPileStack, PT:=T#2S);
	tp_EjectRejectStack(IN:=Stacker.Commands.xEjectRejectStack, PT:=T#2S);

	IF Stacker.Parameters.LineStatusSummary.xEmptyingBelts OR tp_CleanBelts.Q THEN Stacker.Outputs.xCleanBelts := TRUE; END_IF //Not using "tp_CleanBelts.Q"This output must be active all the time since command is received. Disabled when stop button pressed
	IF tp_EjectPileStack.Q THEN Stacker.Outputs.xStackEject := TRUE; END_IF
	IF tp_EjectRejectStack.Q AND Stacker.Parameters.Hw.xRejectEjectionAvailable THEN Stacker.Outputs.xEjectRejectStack := TRUE; END_IF

	//Fall down the commands
	Stacker.Commands:=ResetCommands;

END_PROGRAM
```

#### Status.st
```iecst
ACTION Status:

	CASE Stacker.Status.DeviceStatus OF
		STACKER_TURNED_OFF:
			IF Stacker.Inputs.xStackerPresent THEN
				Stacker.Status.DeviceStatus:=STACKER_INIT;
			END_IF

		STACKER_INIT:
			xBeltsAreStopped:=FALSE;
			IF Stacker.Outputs.xPrepareToStack THEN
				Stacker.Status.DeviceStatus:=STACKER_PREPARING;
			END_IF

		STACKER_PREPARING:
			IF Stacker.Inputs.xReadyToStack THEN
				Stacker.Status.DeviceStatus:=STACKER_READY;
			ELSIF NOT Stacker.Outputs.xPrepareToStack THEN
				Stacker.Status.DeviceStatus:=STACKER_INIT;
			END_IF

		STACKER_READY:
			IF Stacker.Inputs.xRunning THEN
				Stacker.Status.DeviceStatus:=STACKER_WORKING;
			ELSIF NOT Stacker.Inputs.xReadyToStack THEN
				Stacker.Status.DeviceStatus:=STACKER_INIT;
			END_IF

		STACKER_WORKING:
			IF NOT Stacker.Inputs.xRunning THEN
				IF Stacker.Outputs.xRun THEN
					//CapsCases: Stacker stops sometimes due to faulty signal wiring on pdc side. To set faulted state when this occurs so line will stop.
					xBeltsAreStopped:=TRUE;
					Stacker.Status.DeviceStatus:=STACKER_FAULTED;
				ELSE
					Stacker.Status.DeviceStatus:=STACKER_READY;
				END_IF
			END_IF

		STACKER_FAULTED:
			IF NOT Stacker.Inputs.xError THEN
				Stacker.Status.DeviceStatus:=STACKER_INIT;
			END_IF

	END_CASE

	IF NOT Stacker.Inputs.xStackerPresent THEN
		Stacker.Status.DeviceStatus:=STACKER_TURNED_OFF;
	END_IF
	IF Stacker.Status.DeviceStatus <> STACKER_TURNED_OFF AND Stacker.Inputs.xError THEN
		Stacker.Status.DeviceStatus:=STACKER_FAULTED;
	END_IF

	UpdateStatus;

	//Empty belt status
	tiTimeToEmpty := REAL_TO_TIME(60 * (Stacker.Parameters.Hw.rStackerLength + Stacker.Parameters.rMediaLength) / Stacker.Parameters.rSpeedSetPoint);
	tonEmptyBelt.IN := Stacker.Inputs.xRunning;
	tonEmptyBelt.PT := tiTimeToEmpty;
	tonEmptyBelt();
	IF Stacker.Status.Comms.xModuleOk THEN
		Stacker.Status.xBeltEmpty := Stacker.Inputs.Comms.xBeltsEmpty AND NOT Stacker.Inputs.Comms.xStackExit AND (tonEmptyBelt.Q OR NOT Stacker.Inputs.xRunning);
	ELSE
		Stacker.Status.xBeltEmpty := (tonEmptyBelt.Q OR NOT Stacker.Inputs.xRunning);
	END_IF

END_ACTION

ACTION UpdateStatus:

	Stacker.Status.Device.xTurnedOff 	:=	Stacker.Status.DeviceStatus=STACKER_TURNED_OFF;
	Stacker.Status.Device.xInit 		:=	Stacker.Status.DeviceStatus=STACKER_INIT;
	Stacker.Status.Device.xPreparing 	:=	Stacker.Status.DeviceStatus=STACKER_PREPARING;
	Stacker.Status.Device.xReadyToStack	:=	Stacker.Status.DeviceStatus=STACKER_READY;
	Stacker.Status.Device.xStacking 	:=	Stacker.Status.DeviceStatus=STACKER_WORKING;
	Stacker.Status.Device.xFaulted 		:=	Stacker.Status.DeviceStatus=STACKER_FAULTED;

END_ACTION
```

#### StackerCtrl.var - Local variables
```iecst
VAR
	Stacker : REFERENCE TO Stacker_typ;
	AlarmsReseted : StackerAlarms_typ;
	ResetCommands : StackerCommands_typ;
	CommsReset : StackerCommsInputs_typ;
	OutputsReset : StackerOutputs_typ;
	iStackerModel : USINT;
	tp_EjectPileStack : TP;
	tp_EjectRejectStack : TP;
	tp_CleanBelts : TP;
	iIndexHistory : USINT;
	StateHistory : ARRAY[0..iHistoryLines] OF StackerCtrlStatus_enum;
	rMediaThickness : REAL;
	iMinStackBoards : INT := 15; (*Number of minimum boards to be stacked, for both modes: heigh and num of boards*)
	xBeltsAreStopped : BOOL;
END_VAR
VAR CONSTANT
	iHistoryLines : USINT := 20;
END_VAR
VAR
	ModSlaveState : UINT;
	LastError : UINT;
	LastErrorBlockNum : UINT;
	CopyOfWriteData : ARRAY[1..25] OF UINT;
	tonDisableWrittingOfData : TON;
	xDisableWriteData : BOOL;
	ton_CommsError : TON;
	tiTimeToEmpty : TIME;
	tonEmptyBelt : TON;
	EraseWriteData : ARRAY[1..25] OF UINT;
	ton_ControlStopping : TON;
END_VAR
```

### StackerSim.typ
```iecst
TYPE
	StackerSimCommands_typ : 	STRUCT
		StopBelts : BOOL;
		CreateError : BOOL;
	END_STRUCT;
	StackerSim_typ : 	STRUCT
		Commands : StackerSimCommands_typ;
	END_STRUCT;
END_TYPE
```

### StackerSim.var
```iecst
VAR
	SimStacker : REFERENCE TO StackerSim_typ;
	Stacker : REFERENCE TO Stacker_typ;
	tonReady : TON;
	tonRun : TON;
END_VAR
```

### Program Logical/ExtPack/_Ancillaries/SarmCtrl/SarmCtrl/SarmCtrl (IEC)

#### Sarm.st - Init, cyclic, exit code
```iecst
PROGRAM _CYCLIC

	Sarm ACCESS ADR(gSarm);

	//Version
	Sarm.Status.Version.iVersion0 := Sarm.Inputs.Comms.iVersion1;
	Sarm.Status.Version.iVersion1 := Sarm.Inputs.Comms.iVersion2;
	Sarm.Status.Version.iVersion2 := Sarm.Inputs.Comms.iVersion3;
	Sarm.Status.Version.iVersion3 := Sarm.Inputs.Comms.iVersion4;

	//Model evaluation
	iSarmModel.0 := Sarm.Inputs.xModelInput[0];
	iSarmModel.1 := Sarm.Inputs.xModelInput[1];
	iSarmModel.2 := Sarm.Inputs.xModelInput[2];

	Sarm.Status.xInstalled := Sarm.Parameters.xInstalled AND iSarmModel>0;

	//Specify Type of Sarm Model
	Sarm.Status.iModel := iSarmModel;
	CASE iSarmModel OF
		1: Sarm.Status.SarmType := SARMTY_V1;
		ELSE Sarm.Status.SarmType := SARMTY_UNDEFINED;
	END_CASE

	IF NOT Sarm.Status.xInstalled OR NOT Sarm.ParSw.xEnabled THEN
		ResetAlarms;
		Sarm.Outputs := OutputsReset;
		Sarm.Commands:=ResetCommands;
		Sarm.Status.DeviceStatus:=Sarm_TURNED_OFF;
		CopyOfWriteData := EraseWriteData;
		UpdateStatus;
		RETURN;
	END_IF

	IF Sarm.Commands.xResetAlarms THEN ResetAlarms; END_IF

	Configuration;

	Status;

	IF NOT Sarm.Parameters.xSimulationMode THEN
		AssignDataComms;
	END_IF

	//Erasing data when ancillary not in remote
	IF NOT Sarm.Inputs.Comms.xRemote THEN
		CopyOfWriteData := EraseWriteData;
	END_IF

	Alarms;

	IF Sarm.Status.Device.xFaulted OR Sarm.Status.Device.xTurnedOff OR NOT Sarm.Parameters.xLineInAuto THEN
		Sarm.Status.CtrlStatus:=SARMCTRL_STOPPED;
	END_IF

	CASE Sarm.Status.CtrlStatus OF
		SARMCTRL_STOPPED:
			Sarm.Outputs := OutputsReset;
			IF Sarm.Status.DeviceStatus=Sarm_INIT AND Sarm.Commands.xStart THEN
				Sarm.Status.CtrlStatus:=SARMCTRL_STARTING;
			END_IF

		SARMCTRL_STOPPING:
			//Actions
			Sarm.Outputs := OutputsReset;

			Sarm.Outputs.xFastStop := TRUE;

			//Transition
			IF Sarm.Status.DeviceStatus=Sarm_TURNED_OFF OR Sarm.Status.DeviceStatus=Sarm_INIT OR Sarm.Status.DeviceStatus=Sarm_READY THEN
				Sarm.Status.CtrlStatus:=SARMCTRL_STOPPED;
			END_IF

		SARMCTRL_CONTROLSTOPPING:
			//Wait to have the belt empty and send the Stop order
			IF (Sarm.Status.xBeltEmpty AND EDGEPOS(Sarm.Orders.xDisableReadBlock)) OR NOT Sarm.Inputs.xRunning THEN
				Sarm.Status.CtrlStatus:=SARMCTRL_STOPPING;
			END_IF

		SARMCTRL_STARTING:
			//Actions
			Sarm.Outputs.xStartTransport:=TRUE;

			//Transition
			IF Sarm.Status.DeviceStatus=Sarm_READY THEN
				Sarm.Status.CtrlStatus:=SARMCTRL_RUNNING;
			END_IF

		SARMCTRL_RUNNING:
			IF Sarm.Commands.xPause THEN
				Sarm.Status.CtrlStatus:=SARMCTRL_PAUSING;
			END_IF

		SARMCTRL_PAUSING:
			IF Sarm.Status.xBeltEmpty THEN
				//Transition
				Sarm.Status.CtrlStatus:=SARMCTRL_PAUSED;
			END_IF

		SARMCTRL_PAUSED:
			IF Sarm.Commands.xStart THEN
				Sarm.Status.CtrlStatus:=SARMCTRL_STARTING;
			END_IF

	END_CASE

	IF Sarm.Commands.xStop THEN
		Sarm.Status.CtrlStatus:=SARMCTRL_STOPPING;
	ELSIF Sarm.Commands.xControlStop THEN
		Sarm.Status.CtrlStatus:=SARMCTRL_CONTROLSTOPPING;
	END_IF

	//Store the history of the status to easy the debug
	IF Sarm.Status.CtrlStatus<>StateHistory[0] THEN
		FOR iIndexHistory:=iHistoryLines TO 1 BY -1 DO
			StateHistory[iIndexHistory]:=StateHistory[iIndexHistory-1];
		END_FOR
		StateHistory[0]:=Sarm.Status.CtrlStatus;
	END_IF

	Sarm.Commands:=ResetCommands;

END_PROGRAM
```

#### Status.st
```iecst
ACTION Status:

	CASE Sarm.Status.DeviceStatus OF
		Sarm_TURNED_OFF:
			IF Sarm.Inputs.xPowered THEN
				Sarm.Status.DeviceStatus:=Sarm_INIT;
			END_IF

		Sarm_INIT:
			IF Sarm.Outputs.xStartTransport THEN
				Sarm.Status.DeviceStatus:=Sarm_PREPARING;
			END_IF

		Sarm_PREPARING:
			IF Sarm.Inputs.xRunning THEN
				Sarm.Status.DeviceStatus:=Sarm_READY;
			ELSIF NOT Sarm.Outputs.xStartTransport THEN
				Sarm.Status.DeviceStatus:=Sarm_INIT;
			END_IF

		Sarm_READY:
			IF NOT Sarm.Inputs.xRunning THEN
				Sarm.Status.DeviceStatus:=Sarm_INIT;
			END_IF

		Sarm_FAULTED:
			IF NOT Sarm.Inputs.xError THEN
				Sarm.Status.DeviceStatus:=Sarm_TURNED_OFF;
			END_IF

	END_CASE

	IF NOT Sarm.Inputs.xPowered THEN
		Sarm.Status.DeviceStatus:=Sarm_TURNED_OFF;
	END_IF
	IF Sarm.Status.DeviceStatus <> Sarm_TURNED_OFF AND Sarm.Inputs.xError THEN
		Sarm.Status.DeviceStatus:=Sarm_FAULTED;
	END_IF

	UpdateStatus;

	//Empty belt status
	tiTimeToEmpty := REAL_TO_TIME(60 * (Sarm.Parameters.Hw.rSarmLength + Sarm.Parameters.rMediaLength) / Sarm.Parameters.rSpeedSetPoint);
	tonEmptyBelt.IN := Sarm.Inputs.xRunning;
	tonEmptyBelt.PT := tiTimeToEmpty;
	tonEmptyBelt();
	IF Sarm.Status.Comms.xModuleOk THEN
		Sarm.Status.xBeltEmpty:=Sarm.Inputs.Comms.xBeltEmpty AND (tonEmptyBelt.Q OR NOT Sarm.Inputs.xRunning);
	ELSE
		Sarm.Status.xBeltEmpty := (tonEmptyBelt.Q OR NOT Sarm.Inputs.xRunning);
	END_IF

END_ACTION

ACTION UpdateStatus:

	Sarm.Status.Device.xTurnedOff 	:=	Sarm.Status.DeviceStatus=Sarm_TURNED_OFF;
	Sarm.Status.Device.xInit 		:=	Sarm.Status.DeviceStatus=Sarm_INIT;
	Sarm.Status.Device.xPreparing 	:=	Sarm.Status.DeviceStatus=Sarm_PREPARING;
	Sarm.Status.Device.xReady		:=	Sarm.Status.DeviceStatus=Sarm_READY;
	Sarm.Status.Device.xFaulted 	:=	Sarm.Status.DeviceStatus=Sarm_FAULTED;

END_ACTION
```

#### Configuration.st
```iecst
ACTION Configuration:

	CASE Sarm.Status.SarmType OF
		SARMTY_V1:
			// Initial values from OMM-00218_Nozomi_18000+_LED_SARM_Reference_Guide_E1 Document
			Sarm.Parameters.Hw.iMaxMediaWidth := 1800;
			Sarm.Parameters.Hw.iMaxMediaLength := 3200;
			Sarm.Parameters.Hw.iMinMediaThickness := 2;
			Sarm.Parameters.Hw.iMaxMediaThickness := 350;
			Sarm.Parameters.Hw.rSarmLength 	:= 3500;
			Sarm.Parameters.Hw.xDoubleLineAllowed := FALSE;
	END_CASE

END_ACTION
```

#### AssignDataComms.st
```iecst
ACTION AssignDataComms:
	//Active modbus slave diagnosis when ancillary is enabled. This parameter must remain to TRUE from then on.
	//Just would be set to FALSE via UaExpert, to reset historic errors when ancillary is disabled
	Sarm.Parameters.xActiveSlaveDiagnosis := TRUE;

	/////////////////
	//Pre bits treatment
	Sarm.Outputs.Comms.iControl.0 := 	Sarm.Parameters.LineState = LINE_PREPARING_EMPTYBELT OR
										Sarm.Parameters.LineState = LINE_STARTING_EMPTYBELT OR
										Sarm.Parameters.LineState = LINE_BELT_EMPTYING;;

	//Write Registers
	gToWriteDataModbSarm[1] := REAL_TO_UINT(Sarm.Parameters.Media.rLength*10);
	gToWriteDataModbSarm[2] := REAL_TO_UINT(Sarm.Parameters.Media.rWidth*10);
	gToWriteDataModbSarm[3] := REAL_TO_UINT(Sarm.Parameters.Media.rThickness*10);
	gToWriteDataModbSarm[4] := Sarm.Parameters.iLineConfig; //REAL_TO_UINT(Sarm.Parameters.Media.rGap*10);
//	gToWriteDataModbSarm[5] := ;
//	gToWriteDataModbSarm[6] := ;
	gToWriteDataModbSarm[7] := REAL_TO_UINT(Sarm.Parameters.rSpeedSetPoint*10);
	gToWriteDataModbSarm[8] := Sarm.Outputs.Comms.iControl;

	//Disabling writting after some time active. To test
	tonDisableWrittingOfData.IN:= NOT xDisableWriteData;
	tonDisableWrittingOfData.PT:= T#1000ms;
	tonDisableWrittingOfData();

	IF tonDisableWrittingOfData.Q THEN
		xDisableWriteData := TRUE;
	END_IF

	FOR iIndex:=1 TO 25 DO
		IF gToWriteDataModbSarm[iIndex]<>CopyOfWriteData[iIndex] THEN
			xDisableWriteData := FALSE;
		END_IF
	END_FOR

	Sarm.Orders.xDisableWriteBlock := xDisableWriteData;

	//Copying previous data
	CopyOfWriteData := gToWriteDataModbSarm;

	////////////////
	//Read Registers
	IF Sarm.Status.Comms.xModuleOk THEN
		Sarm.Inputs.Comms.iStatus := gReceivedDataModbSarm[1]; // Status Word
		Sarm.Inputs.Comms.iAlarmWord1 := gReceivedDataModbSarm[2]; // Alarm word 1 - Critical alarms
		Sarm.Inputs.Comms.iAlarmWord2 := gReceivedDataModbSarm[3]; // Alarm word 2
		Sarm.Inputs.Comms.iAlarmWord3 := gReceivedDataModbSarm[4]; // Alarm word 3
		//		Sarm.Inputs.Comms. := gReceivedDataModbSarm[5]; //Review SARM code to understand what information is being shared
		//		 := gReceivedDataModbSarm[6];
		//		 := gReceivedDataModbSarm[7];
		//		:= gReceivedDataModbSarm[8];
		//		:= gReceivedDataModbSarm[9];
		Sarm.Inputs.Comms.iVersion1 := gReceivedDataModbSarm[10];
		Sarm.Inputs.Comms.iVersion2 := gReceivedDataModbSarm[11];
		Sarm.Inputs.Comms.iVersion3 := gReceivedDataModbSarm[12];
		Sarm.Inputs.Comms.iVersion4 := gReceivedDataModbSarm[13];
		//		 := gReceivedDataModbSarm[14];
		//		 := gReceivedDataModbSarm[15];

	END_IF

	//Post bit treatment
	Sarm.Inputs.Comms.xRemote := Sarm.Inputs.Comms.iStatus.0;
	Sarm.Inputs.Comms.xAlarmPresent := Sarm.Inputs.Comms.iStatus.1;
	Sarm.Inputs.Comms.xBeltEmpty := Sarm.Inputs.Comms.iStatus.2; //Not being written on SARM code (FALSE assignation in that code)
	Sarm.Inputs.Comms.xWarningPresent := Sarm.Inputs.Comms.iStatus.3;
	Sarm.Inputs.Comms.xOnline := Sarm.Inputs.Comms.iStatus.4;
	Sarm.Inputs.Comms.xSafetyOnline := Sarm.Inputs.Comms.iStatus.5;

END_ACTION
```

### Program Logical/ExtPack/_Ancillaries/SarmCtrl/SarmSim/SarmSim_v1/SarmSim (IEC)

#### SarmSim.st - Init, cyclic, exit code
```iecst
PROGRAM _INIT

	Sarm ACCESS ADR(gSarm);
	SimSarm ACCESS ADR(gSimSarm);

	Sarm.Status.Comms.xModuleOk := TRUE;

END_PROGRAM

PROGRAM _CYCLIC
	(* Insert code here *)
	Sarm ACCESS ADR(gSarm);
	SimSarm ACCESS ADR(gSimSarm);

	Sarm.Inputs.xSarmPresent := TRUE;
	Sarm.Inputs.Comms.xOnline := TRUE;
	Sarm.Inputs.Comms.xRemote := TRUE;
	Sarm.Inputs.xPowered := TRUE;
	Sarm.Inputs.xError:=SimSarm.Commands.CreateError;

	tonPrepare.IN:=	Sarm.Outputs.xStartTransport;
	tonPrepare.PT:= T#2s;
	tonPrepare();
	Sarm.Inputs.xRunning:=tonPrepare.Q;

	Sarm.Inputs.Comms.iVersion1 := 1;
	Sarm.Inputs.Comms.iVersion2 := 1;
	Sarm.Inputs.Comms.iVersion3 := 3;
	Sarm.Inputs.Comms.iVersion4 := 15;

	Sarm.Inputs.Comms.xBeltEmpty := TRUE;

END_PROGRAM
```

### SarmSim.typ
```iecst
TYPE
	SarmSimCommands_typ : 	STRUCT
		CreateError : BOOL;
	END_STRUCT;
	SarmSim_typ : 	STRUCT
		Commands : SarmSimCommands_typ;
	END_STRUCT;
END_TYPE
```

### Program Logical/ExtPack/_Cure/CuringLedCtrl/CuringLedCtrl_v1/InitCuringLedCtrl (IEC)

#### InitCuringLedCtrl.st - Init, cyclic, exit code
```iecst
PROGRAM _CYCLIC
	iIndexCuringLed := 1;
END_PROGRAM
```

### Program Logical/ExtPack/_Cure/CuringLedCtrl/CuringLedCtrl_v1/CuringLedCtrl (IEC)

#### CuringLedCtrl.st - Init, cyclic, exit code
```iecst
PROGRAM _INIT
	NitroState := CURINGNITRO_OFF;
END_PROGRAM

PROGRAM _CYCLIC

	//References of the program
	dataLed 	ACCESS ADR (gCuringLed[iIndexCuringLed]);
	dataChiller	ACCESS ADR (gChiller[gCuringLed[iIndexCuringLed].Parameters.iChillerIndex]);

	dataLed.Status.xCureByStretch := dataLed.Parameters.xCureByStretch;
	dataLed.Status.xOptimizeCuring := dataLed.Parameters.xOptimizeCuring;
	dataLed.Status.xInstalled := dataLed.Parameters.xInstalled;
	dataLed.Status.ChillerState := dataChiller.St.Status;

	IF NOT dataLed.Parameters.xInstalled THEN
		ResetAlarms;
		ResetOutputs;
		iIndexCuringLed:= iIndexCuringLed +1;
		RETURN;
	END_IF

	//Reset alarms
	IF dataLed.Commands.Reset THEN
		ResetAlarms;
	END_IF

	CheckParameters;

	StateManager;
	StateNitrogen;

	//////	    CuringByStretch		//////
	//Serial Comms
	xAnyParamChanged.0 := iPreviousWidth <> dataLed.Status.iCuringAreaWidth;
	xAnyParamChanged.1 := iPreviousOffsetRegisterL1 <> dataLed.Status.iCuringAreaOffsetL1;
	xAnyParamChanged.2 := iPreviousOffsetRegisterL2 <> dataLed.Status.iCuringAreaOffsetL2;
	xAnyParamChanged.3 := EDGEPOS(dataLed.Status.xLampsDetected);
	xAnyParamChanged.4 := EDGEPOS(tonLampsVoltageRecovery.Q);
	xBoardPositionChanged := (dataLed.Status.iCuringAreaWidth>=0) AND (xAnyParamChanged > 0);

	IF xBoardPositionChanged THEN
		StretchesCalculation; //To execute this action to calculate basic parameters
		EnableLamps;

		IF dataLed.Status.xCureByStretch THEN
			//Calculation of lamps SLM (sections) to be enabled
			IF NOT dataLed.Parameters.xDoubleLine THEN SingleLineCalculation; ELSE DoubleLineCalculation; END_IF
		END_IF

		//To save current board position and width values
		MemoBoardParameters;
	END_IF

	//To evaluate if detect lamps action must be executed in case curing by stretch is enabled
	IF EDGEPOS(dataLed.Parameters.xCureByStretch) THEN
		//To reset lamp's serial numbers
		FOR iIndexDetectLamps:=1 TO iLampsQuantity DO
			IF (dataLed.Lamp[iIndexDetectLamps].Status.stSerialNumber = '') THEN dataLed.Status.xLampsDetected := FALSE; END_IF
		END_FOR
	END_IF

	DetectLamps;
	IF dataLed.Status.xLampsDetected THEN
		//Curing by stretch
		IF dataLed.Status.xCureByStretch THEN
			//Execute lamp's SLMs config
			ConfigureLamps;
			CheckLampsConfig;
		END_IF

		//Getting useful information from lamps
		IF NOT dataLed.Parameters.xPhysicalTempFeedback THEN
			ReadTemperature;
		END_IF

		//ReadUvOnTime;

	END_IF

	//Comms management
	CommsManager;

	//DELOREAN-1521: To switch on curing subsystems but not active alarms while not enabled
	IF dataLed.Parameters.xEnabled OR xDetectionLampsProcessOn THEN
		Alarms;
	END_IF

	//Alarm Sound
	AlarmSound;

	//OUTPUTS//
	//Defining setting previous to call action to set intensity
	IF dataLed.Parameters.CuringApplicationType = CURING_APP_WHITE THEN
		rCureBySpeedSlope := rCureBySpeedWhiteSlope;
		rCureBySpeedIntercept := rCureBySpeedWhiteIntercept;
	ELSE
		//[RGP] Pending to consider parameter "Primer" instead of color but till defined, this curing bar will use "Color" information
		rCureBySpeedSlope := rCureBySpeedDefaultSlope;
		rCureBySpeedIntercept := rCureBySpeedDefaultIntercept;
	END_IF

	//Setting intensity
	SetLampsIntensity;

	//Detection state
	dataLed.Status.xLampsDetected := DetectStep = DETECTION_READY;

	//Chiller
	dataLed.Signals.Outputs.xRunChiller := dataLed.Commands.RunCuring OR dataLed.Commands.xRunNitrogenFlow;

	//Nitrogen
	dataLed.Signals.Outputs.xPowerOnNitrogen := //Manual
												dataLed.Commands.Manual.xNitrogen OR
												//Auto
												dataLed.Commands.xRunNitrogenFlow;

	//Curing lamp's power supply management
	//DELOREAN-962: QA wants lamps to be powered after some time instead of wait to press reset to remove alarms
	tonPowerOnLamps(IN:=NOT dataLed.Signals.Outputs.xPowerOnLamps, PT:=T#10s);
	IF EDGENEG(dataLed.Status.xCureByStretch) OR (dataLed.Commands.Manual.ResetPSU) OR NOT xPowerOnLamps THEN
		dataLed.Signals.Outputs.xPowerOnLamps := FALSE;
	ELSE
		IF (tonPowerOnLamps.Q) THEN
			dataLed.Signals.Outputs.xPowerOnLamps := TRUE;
		END_IF
	END_IF

	//Copying outputs related to manual commands
	dataLed.Status.ManualCommands.xNitrogen := dataLed.Signals.Outputs.xPowerOnNitrogen;

	//Resetting manual commands
	//To reset manual commands when not in manual mode
	IF NOT dataLed.Parameters.Mode.xManual THEN dataLed.Commands.Manual := ResetManCommands; END_IF

	//Prepare for the next element
	iIndexCuringLed:= iIndexCuringLed +1;

END_PROGRAM
```

#### StateNitrogen.st
```iecst
ACTION StateNitrogen:

	CASE NitroState OF

		CURINGNITRO_OFF:
			IF StatusCtrl <> CURINGLED_OFF THEN
				NitroState := CURINGNITRO_INIT;
			END_IF

		CURINGNITRO_INIT:
			IF dataLed.Signals.Outputs.xPowerOnNitrogen THEN
				NitroState := CURINGNITRO_READY;
			END_IF

		CURINGNITRO_FAULT:
			IF NOT dataLed.Alarms.xN2LowFlow THEN
				NitroState := CURINGNITRO_READY;
			END_IF

		CURINGNITRO_READY:
			//[RGP] Line status considered due to issue NOZOMI-16649. Nitrogen low flow alarm will execute a controlled stop, but curing wont stop till line has stopped
			IF dataLed.Alarms.xN2LowFlow AND NOT dataLed.Commands.xRunNitrogenFlow THEN
				NitroState := CURINGNITRO_FAULT;
			END_IF

	END_CASE

	IF StatusCtrl = CURINGLED_OFF  THEN
		NitroState := CURINGNITRO_OFF;
	END_IF

	dataLed.Status.NitroState:=NitroState;

END_ACTION
```

#### DetectLamps.st
```iecst
ACTION DetectLamps:

	//Command to look for serial numbers
	IF EDGEPOS (dataLed.Commands.Manual.DetectLamps) THEN
		DetectStep := DETECTION_INIT;
		dataLed.Commands.Manual.DetectLamps := FALSE;
		dataLed.Comms.Command.Close := TRUE;
	END_IF

	//Timer to end FinishPolling step as a redundancy
	tonFinishPolling.IN := DetectStep = DETECTION_FINISHING_POLLING;
	tonFinishPolling.PT := T#30s;
	tonFinishPolling();

	CASE DetectStep OF

		DETECTION_NOT_INIT:
			//dataLed.Comms.Command.Close := TRUE; //[RGP]DELOREAN-1136. Close command executed in error state

		DETECTION_INIT:
			iIndexDetectLamps := 0;
			iIndexPreSerialNumbers := 1;

			//To reset lamp's serial numbers
			FOR iIndexDetectLamps:=1 TO iLampsQuantity DO
				dataLed.Lamp[iIndexDetectLamps].Status.stSerialNumber := '';
			END_FOR

			//To reset array of PreSerial numbers
			FOR i:=1 TO 15 DO
				aPreSerialNumbers[i] := '';
			END_FOR

			dataLed.Comms.Device.receive_data := '';
			DetectStep := DETECTION_POLLING;

		DETECTION_POLLING:
			Poll;

			IF (StAnswer<>'') THEN
				DetectStep := DETECTION_SAVE_SERIAL_NUMBERS;
			ELSIF dataLed.Comms.Device.step = FRM_WAIT THEN
				//To send command to lamp
				dataLed.Comms.Command.Send := TRUE;
			END_IF

		DETECTION_SAVE_SERIAL_NUMBERS:
			IF iIndexPreSerialNumbers <= iLampsQuantity THEN
				//Every time a poll message is sent, device writes one serial number
				//[RGP] 'Custom' is a message that lamps sends every x seconds so sometimes was being save as a valid serial number.
				IF (StAnswer <> '') AND (StAnswer <> 'Custom') THEN
					StMessage:='';
					xRepeated := FALSE;
					FOR iIndexDetectLamps:=1 TO iLampsQuantity DO
						IF (StAnswer = aPreSerialNumbers[iIndexDetectLamps]) THEN xRepeated := TRUE; END_IF
					END_FOR

					IF NOT xRepeated THEN
						aPreSerialNumbers[iIndexPreSerialNumbers] := StAnswer;
						iIndexPreSerialNumbers := iIndexPreSerialNumbers + 1;
					ELSE
						dataLed.Comms.Device.receive_data := '';
					END_IF

				ELSIF (dataLed.Comms.Device.step = FRM_WAIT)THEN
					//To send command to lamp
					dataLed.Comms.Command.Send := TRUE;
				END_IF
			ELSE
				dataLed.Comms.Device.receive_data := '';
				iIndexPreSerialNumbers := 1;
				DetectStep := DETECTION_FINISHING_POLLING; //DETECTION_READ_INTENSITY;
			END_IF

		DETECTION_FINISHING_POLLING:
			//StMessage:='';
			ReadFinishPolling;
			IF (StAnswer=StGoodAnswer OR tonFinishPolling.Q) THEN
				dataLed.Comms.Command.Close := TRUE;
				dataLed.Comms.Device.receive_data := '';
				DetectStep := DETECTION_READ_INTENSITY;
			ELSIF (dataLed.Comms.Device.step = FRM_WAIT) THEN
				//To send command to lamp
				dataLed.Comms.Command.Send := TRUE;
			END_IF

		DETECTION_READ_INTENSITY:
			ReadLampIntensity;

			IF (StAnswerAux='0') THEN
				DetectStep := DETECTION_ASSIGN_POSITION;
			ELSIF (dataLed.Comms.Device.step = FRM_WAIT)THEN
				//To send command to lamp
				dataLed.Comms.Command.Send := TRUE;
			END_IF

		DETECTION_ASSIGN_POSITION:
			IF iIndexPreSerialNumbers <= iLampsQuantity THEN

				//To assign a pre serial number saved to its lamp
				iDetectedLamp := STRING_TO_INT(StAnswer); //Convert number extracted from intensity, which match lamp position, to an INT to do the assignation
				IF (iDetectedLamp <= iLampsQuantity) THEN
					IF (dataLed.Lamp[iDetectedLamp].Status.stSerialNumber = '') THEN
						dataLed.Lamp[iDetectedLamp].Status.stSerialNumber := aPreSerialNumbers[iIndexPreSerialNumbers];
					END_IF
				END_IF

				//To know whether all lamps have a serial number assigned
				xKeepFilling := FALSE;
				FOR iIndexDetectLamps:=1 TO iLampsQuantity DO
					IF (dataLed.Lamp[iIndexDetectLamps].Status.stSerialNumber = '') THEN
						xKeepFilling := TRUE;
					END_IF
				END_FOR

				//All lamps have a SN assigned
				IF NOT xKeepFilling THEN
					iDetectLampAttempts := 0;
					DetectStep := DETECTION_READY;

				//Exceeded max number of attempts to find as serial numbers as quantity of lamps installed. To review RS485 wiring
				ELSIF iDetectLampAttempts >= iMaxNumAttempts OR iIndexPreSerialNum>iLampsQuantity THEN
					iDetectLampAttempts := 0;
					iIndexPreSerialNum := 1;
					dataLed.Comms.Device.receive_data := '';

				//To check next preSN saved
				ELSE
					iIndexPreSerialNumbers := iIndexPreSerialNumbers + 1;
					dataLed.Comms.Device.receive_data := '';
					DetectStep := DETECTION_READ_INTENSITY;
				END_IF
			END_IF

		DETECTION_READY:

		DETECTION_ERROR:
			dataLed.Comms.Command.Close := TRUE;
			IF dataLed.Commands.Reset THEN DetectStep := DETECTION_NOT_INIT; END_IF

	END_CASE

	//Process is cancelled in case machine mode goes out of manual and process were not finished or in error
	IF (NOT dataLed.Parameters.Mode.xManual) AND (DetectStep <> DETECTION_READY) AND (DetectStep <> DETECTION_ERROR) THEN
		DetectStep := DETECTION_ERROR; //[RGP]DELOREAN-1136: To set ERROR state when this conditions occur and then when reset command is received, go to NOT_INIT
	END_IF

	dataLed.Comms.Device.send_data := StMessage; //To assign Message to dataled comms struct
	StAnswer := MID(dataLed.Comms.Device.receive_data, iAnswerStringLength, iAnswerStringPosition);
	StAnswerAux := MID(dataLed.Comms.Device.receive_data, iAnswerStringLength, 1);
	dataLed.Status.DetectionState := DetectStep;

	xDetectionLampsProcessOn := (DetectStep <> DETECTION_NOT_INIT) AND
								(DetectStep <> DETECTION_READY) AND
								(DetectStep <> DETECTION_ERROR);

END_ACTION

ACTION Poll:
	//To define the string to be sent to the lamp
	StMessage := StPoll;
	iAnswerStringPosition := 1;
	iAnswerStringLength := 6;
END_ACTION

//Telegrams to be sent to curing led devices//
//To read lamp's intensity setpoint
ACTION ReadLampIntensity:
	//To define the string to be sent to the lamp
	StMessage := StCmdRead;
	//strcat: Used to link (concat) several strings
	strcat(ADR(StMessage), ADR(aPreSerialNumbers[iIndexPreSerialNumbers]));
	strcat(ADR(StMessage), ADR(StMl));
	strcat(ADR(StMessage), ADR(StIntensity));

	//Devices answers a number
	StGoodAnswer := INT_TO_STRING(iIndexDetectLamps);

	iAnswerStringPosition := 2;
	iAnswerStringLength := 1;
	//This is the data received when reading lamp's intensity: 10% = 010; 25%=025; 99%=099

END_ACTION

ACTION ReadFinishPolling:
	//To define the string to be sent to the lamp
	StMessage := '';

	//Devices answers a number
	StGoodAnswer := 'Custom';

	iAnswerStringPosition := 1;
	iAnswerStringLength := 6;
	//This is the data received when reading lamp's intensity: 10% = 010; 25%=025; 99%=099

END_ACTION
```

#### Alarms.st
```iecst
ACTION Alarms:

	IF dataLed.Status.State = CURINGLED_FAULTED THEN
		dataLed.Alarms.xCureSystemFaulted := TRUE;
	END_IF

	dataLed.Alarms.xChillerFaulted := dataChiller.St.Status = CHILLER_FAULT;

	IF dataLed.Signals.Inputs.xN2HighFlow AND dataLed.Signals.Outputs.xPowerOnNitrogen THEN
		dataLed.Alarms.xN2HighFlow := TRUE;
	END_IF

	tonNitroAlrLowFlow.IN := dataLed.Signals.Inputs.xN2LowFlow AND dataLed.Signals.Outputs.xPowerOnNitrogen;
	tonNitroAlrLowFlow.PT := T#4s;
	tonNitroAlrLowFlow();
	IF tonNitroAlrLowFlow.Q THEN
		dataLed.Alarms.xN2LowFlow := TRUE;
	END_IF

	//Assign alarms and create the words with all the alarm bits
	errorLampsSLM:=0;
	errorLampsThermal:=0;

	tonCheckAlarms.IN := dataLed.Signals.Inputs.xSafetyEnable;
	tonCheckAlarms.PT := T#3000ms;
	tonCheckAlarms();

	IF tonCheckAlarms.Q THEN
		FOR iIndexCuring:=1 TO iLampsQuantity DO
			//SLM faults are only critical when led is enabled to cure
			IF dataLed.Lamp[iIndexCuring].Parameters.EnabledByPosition THEN
				dataLed.Alarms.Lamps[iIndexCuring].SLMFault := dataLed.Lamp[iIndexCuring].Inputs.SLMFault;
			ELSE
				dataLed.Alarms.Lamps[iIndexCuring].AnyWarning := dataLed.Lamp[iIndexCuring].Inputs.SLMFault;
			END_IF
			IF dataLed.Alarms.Lamps[iIndexCuring].SLMFault THEN
				errorLampsSLM := errorLampsSLM OR SHL(1,iIndexCuring-1);
			END_IF

			//Thermal faults are always evaluated, either the led is enabled to cure or not
			dataLed.Alarms.Lamps[iIndexCuring].ThermalFault := dataLed.Lamp[iIndexCuring].Inputs.ThermalFault;
			IF dataLed.Alarms.Lamps[iIndexCuring].ThermalFault THEN
				errorLampsThermal := errorLampsThermal OR SHL(1,iIndexCuring-1);
			END_IF
		END_FOR
	END_IF

	//Power supplies
	xPowerOnLamps := TRUE;
	FOR iIndexPowerSupply:=1 TO iPowerSuppliesQuantity DO
		tonStabPsuFailure[iIndexPowerSupply].IN := NOT dataLed.Signals.Inputs.xPsuDcOk[iIndexPowerSupply] OR NOT dataLed.Signals.Inputs.xPsuAcOk[iIndexPowerSupply];
		tonStabPsuFailure[iIndexPowerSupply].PT := T#300ms;
		tonStabPsuFailure[iIndexPowerSupply]();
		IF tonStabPsuFailure[iIndexPowerSupply].Q AND tonCheckAlarms.Q THEN
			IF NOT dataLed.Alarms.xPowerFailure THEN
				LogPsuFailure;
			END_IF
			dataLed.Alarms.xPowerFailure := TRUE;
		END_IF
		IF NOT dataLed.Signals.Inputs.xPsuAcOk[iIndexPowerSupply] THEN
			xPowerOnLamps := FALSE;
		END_IF
	END_FOR

	//Timer to launch lamps configuration after voltage recovery
	tonLampsVoltageRecovery.IN := NOT dataLed.Alarms.xPowerFailure;
	tonLampsVoltageRecovery.PT := T#5s;
	tonLampsVoltageRecovery();

	//Front door opened
	IF NOT dataLed.Signals.Inputs.xFrontDoorClosed AND dataLed.Status.xEmitting THEN
		dataLed.Alarms.xFrontDoorOpened := TRUE;
	END_IF

	//Curing by stretch related
	IF dataLed.Status.xCureByStretch AND NOT dataLed.Parameters.xSimulationMode THEN

		IF EDGEPOS(dataLed.Status.xLampsChecked) THEN //DELOREAN-1814: In case configuration process fails, lamps may be power cycled and then full width is set by job, to not raise this alarm
			xConfigurationFailed := FALSE;
			//Lamp's stretches not configured
			FOR iIndexCheckLamps:=1 TO iLampsQuantity DO
				iNumLampSLM := dataLed.Lamp[iIndexCheckLamps].Parameters.iNumSLM;
				FOR iIndexCheckSlm:=1 TO iNumLampSLM DO
					//To check that SLM activated matches with slms calculated to be enabled
					IF dataLed.Lamp[iIndexCheckLamps].Outputs.xSlmStatus[iIndexCheckSlm] <> dataLed.Lamp[iIndexCheckLamps].Parameters.xSlmEnable[iIndexCheckSlm] THEN
						xConfigurationFailed := TRUE;
						dataLed.Alarms.Lamps[iIndexCheckLamps].xSlmWrongConfiguration[iIndexCheckSlm]:=TRUE;
					ELSE
						dataLed.Alarms.Lamps[iIndexCheckLamps].xSlmWrongConfiguration[iIndexCheckSlm]:=FALSE;
					END_IF
				END_FOR

				//Lamp status feedback error
				//IF dataLed.Alarms.Lamps[iIndexCheckLamps].StatusFeedbackFault THEN xConfigurationFailed := TRUE; END_IF
			END_FOR

		END_IF

		//SlmNotConfigured. Autoreset
		IF xConfigurationFailed THEN
			dataLed.Alarms.xLampsSlmNotConfigured := TRUE; // OR NOT dataLed.Status.xLampsConfigured;
		END_IF

		//Lamps serial number not assigned
		FOR iIndexCuring:=1 TO iLampsQuantity DO
			IF (dataLed.Lamp[iIndexCuring].Status.stSerialNumber = '') THEN
				dataLed.Alarms.xSerialNumbersNotAssigned := TRUE;
			END_IF

			IF dataLed.Status.xLampsDetected THEN
				FOR iIndexCuringAux:=1 TO iLampsQuantity DO
					IF (iIndexCuringAux<>iIndexCuring) AND (dataLed.Lamp[iIndexCuringAux].Status.stSerialNumber = dataLed.Lamp[iIndexCuring].Status.stSerialNumber) THEN
						dataLed.Alarms.xSerialNumbersRepeated := TRUE;
					END_IF
				END_FOR
			ELSE
				dataLed.Alarms.xSerialNumbersRepeated := FALSE;
			END_IF
		END_FOR

		//Detection process has failed
		IF dataLed.Status.DetectionState = DETECTION_ERROR THEN
			dataLed.Alarms.xDetectionProcessFailed := TRUE;
		ELSE
			dataLed.Alarms.xDetectionProcessFailed := FALSE;
		END_IF
	ELSE
		dataLed.Alarms.xLampsSlmNotConfigured := FALSE;
		dataLed.Alarms.xSerialNumbersNotAssigned := FALSE;
		dataLed.Alarms.xDetectionProcessFailed := FALSE;
	END_IF

	// ALARMS SUMMARY
	AlarmsSummary;

END_ACTION

ACTION ResetAlarms:
	dataLed.Alarms := AlarmsReseted;
	dataLed.AlSummary := AlarmsSummaryReseted;
END_ACTION
```

#### AlarmsSummary.st
```iecst
ACTION AlarmsSummary:

	//Alarms Summary
	//Warning
	iReasonWarning.0 := dataLed.Alarms.xN2HighFlow;
	iReasonWarning.1 := dataLed.Alarms.xSerialNumbersRepeated;

	dataLed.AlSummary.xAnyWarning := iReasonWarning > 0;

	//Stop
	iReasonStop.0 := dataLed.Alarms.xN2LowFlow;
	iReasonStop.1 := dataLed.Alarms.xLampsSlmNotConfigured;
	iReasonStop.2 := dataLed.Alarms.xFrontDoorOpened;

	dataLed.AlSummary.xAlarmStop :=	iReasonStop > 0;
	IF EDGEPOS(dataLed.AlSummary.xAlarmStop) THEN
		dataLed.AlSummary.iReasonStop[0] := iReasonStop;
		LogStopAlarm;
	ELSIF EDGEPOS(NOT dataLed.Parameters.AutoMode.xStop AND NOT dataLed.AlSummary.xAlarmStop) THEN
		dataLed.AlSummary.iReasonStop[0] := 0;
	END_IF

	//Critical
	iReasonCritical.0 := dataLed.Alarms.xCureSystemFaulted;
	iReasonCritical.1 := errorLampsSLM>0;
	iReasonCritical.2 := errorLampsThermal>0;
	iReasonCritical.3 := dataLed.Alarms.xSerialNumbersNotAssigned;
	iReasonCritical.4 := dataLed.Alarms.xDetectionProcessFailed;
	iReasonCritical.5 := dataLed.Alarms.xPowerFailure;

	dataLed.AlSummary.xAlarmCritical:= iReasonCritical > 0 AND dataLed.Parameters.Mode.xAuto;
	IF EDGEPOS(dataLed.AlSummary.xAlarmCritical) THEN
		dataLed.AlSummary.iReasonCritical := iReasonCritical;
		LogCriticalAlarm;
	ELSIF EDGEPOS(dataLed.Parameters.Mode.xAuto AND iReasonCritical=0) THEN
		dataLed.AlSummary.iReasonCritical := 0;
	END_IF

END_ACTION
```

#### SetLampsIntensity.st
```iecst
ACTION SetLampsIntensity:

	//Assign the enable and intensity value to the output signals
	xCuringOrder := (StatusCtrl = CURINGLED_EMITTING);
	FOR iIndexCuring:=1 TO iLampsQuantity DO
		//To enable lamp
		dataLed.Lamp[iIndexCuring].Outputs.EnableLamp := xCuringOrder AND dataLed.Lamp[iIndexCuring].Parameters.EnabledByPosition AND dataLed.Parameters.xEnabled;

		IF dataLed.Parameters.xPhysicalTempFeedback THEN
			dataLed.Lamp[iIndexCuring].Outputs.rTemperature := (dataLed.Lamp[iIndexCuring].Inputs.TemperatureRaw/327.7);
		END_IF

		//To set lamp's intensity depending on state mode
		//Auto = Intensity set on the UI
		IF (dataLed.Parameters.rBeltCurrentSpeed<=iMinSpeedWhenBlockAtSafePosition) THEN
			iIntensityWhileAtSafePosition:=30;
		ELSE
			iIntensityWhileAtSafePosition:=40;
		END_IF

		IF dataLed.Parameters.Mode.xAuto THEN
			IF dataLed.Commands.xDropPower THEN
				dataLed.Lamp[iIndexCuring].Outputs.IntensityLampRaw := REAL_TO_INT(iIntensityWhileAtSafePosition * rLampIntensitySlope); //10V correspond to 32766

			ELSIF dataLed.Parameters.xCureBySpeed THEN
				iIntensityCureBySpeed := REAL_TO_USINT((rCureBySpeedSlope * dataLed.Parameters.rBeltCurrentSpeed) + rCureBySpeedIntercept);
				iIntensityCureBySpeed := LIMIT(MinIntensityCuringBySpeed, iIntensityCureBySpeed, MaxIntensityCuringBySpeed);
				dataLed.Lamp[iIndexCuring].Outputs.IntensityLampRaw := REAL_TO_INT(iIntensityCureBySpeed * rLampIntensitySlope); //10V correspond to 32766

			ELSE
				dataLed.Lamp[iIndexCuring].Outputs.IntensityLampRaw := REAL_TO_INT(dataLed.parSw.IntensitySetPoint * rLampIntensitySlope); //10V correspond to 32766
			END_IF

			//Manual = Intensity set by PLC in case of detect lamps process is going on
		ELSIF dataLed.Parameters.Mode.xManual THEN
			IF 	(DetectStep = DETECTION_READ_INTENSITY) OR
				(DetectStep = DETECTION_ASSIGN_POSITION) THEN
				//To multiply by 11 so in case of analogic intensity output is a bit low than desired, we get the number correctly.
				//Example: 1*11=11, will read either 010, 011 or 012. 1 is always the second number. If using 1*10, may get a 009 and no "1" will be found
				dataLed.Lamp[iIndexCuring].Outputs.IntensityLampRaw := REAL_TO_INT(iIndexCuring*11 * rLampIntensitySlope);
			END_IF

			//Zero = Intensity set to zero as a safety redundancy
		ELSE
			dataLed.Lamp[iIndexCuring].Outputs.IntensityLampRaw := 0;
		END_IF

		//Convert raw data to percentage
		dataLed.Lamp[iIndexCuring].Outputs.IntensityLampApplied := REAL_TO_USINT(dataLed.Lamp[iIndexCuring].Outputs.IntensityLampRaw/rLampIntensitySlope);
	END_FOR

END_ACTION

ACTION ResetOutputs:
	dataLed.Signals.Outputs := OutputsReset;
END_ACTION
```

#### ReadTemperature.st
```iecst
ACTION ReadTemperature:

	IF NOT dataLed.Status.xLampsDetected OR (dataLed.Status.xCureByStretch AND NOT dataLed.Status.xLampsChecked) THEN
		ReadingTemperatureStep := READINGTEMP_NOT_INIT;
	END_IF

	CASE ReadingTemperatureStep OF

		READINGTEMP_NOT_INIT:
			iIndexReadTempLamps := 1;
			IF (ReadingUvOnTimeStep = READINGUVTIME_NOT_INIT) THEN
				ReadingTemperatureStep := READINGTEMP_INIT;
			END_IF

		READINGTEMP_INIT:
			dataLed.Comms.Command.Close := TRUE;
			dataLed.Comms.Device.receive_data := '';

			ReadingTemperatureStep := READINGTEMP_READING;

		READINGTEMP_READING:

			ReadLampTemperature;
			StAnswer := MID(dataLed.Comms.Device.receive_data, iAnswerStringLength, iAnswerStringPosition);
			IF (StAnswer<>'') THEN // AND (StAnswerAux<>'') THEN
				ReadingTemperatureStep := READINGTEMP_READY;

			ELSIF (dataLed.Comms.Device.step = FRM_WAIT)THEN
				//To send command to lamp
				dataLed.Comms.Command.Send := TRUE;
			END_IF

		READINGTEMP_READY:

			dataLed.Lamp[iIndexReadTempLamps].Status.rTemp := brsatof(ADR(StAnswer));

			// Assigning value to value assigned if there is an analog card
			dataLed.Lamp[iIndexReadTempLamps].Outputs.rTemperature := dataLed.Lamp[iIndexReadTempLamps].Status.rTemp;

			ReadNextLampTemp;

	END_CASE

	dataLed.Comms.Device.send_data := StMessage;

END_ACTION

//Telegrams to be sent to curing led devices//
//To read lamp's intensity setpoint
ACTION ReadLampTemperature:
	//To define the string to be sent to the lamp
	StMessage := StCmdRead;
	//strcat: Used to link (concat) several strings
	strcat(ADR(StMessage), ADR(dataLed.Lamp[iIndexReadTempLamps].Status.stSerialNumber));
	strcat(ADR(StMessage), ADR(StMl));
	strcat(ADR(StMessage), ADR(StTemperature));

	iAnswerStringLength := 4;
	iAnswerStringPosition := 1;

END_ACTION

ACTION ReadNextLampTemp:

	//Erasing buffer and going to next lamp
	iIndexReadTempLamps := iIndexReadTempLamps + 1;
	IF iIndexReadTempLamps <= iLampsQuantity THEN
		ReadingTemperatureStep := READINGTEMP_INIT;
	ELSE
		ReadingTemperatureStep := READINGTEMP_NOT_INIT;
	END_IF

END_ACTION
```

#### ReadUvOnTime.st
```iecst
ACTION ReadUvOnTime:

	IF NOT dataLed.Status.xLampsDetected OR (dataLed.Status.xCureByStretch AND NOT dataLed.Status.xLampsChecked) OR ReadingTemperatureStep <> READINGTEMP_NOT_INIT THEN
		ReadingUvOnTimeStep := READINGUVTIME_NOT_INIT;
	END_IF

	CASE ReadingUvOnTimeStep OF

		READINGUVTIME_NOT_INIT:
			iIndexReadUvOnTimeLamps := 1;
			IF (NOT dataLed.Parameters.xPhysicalTempFeedback AND EDGEPOS(ReadingTemperatureStep = READINGTEMP_NOT_INIT) OR
				dataLed.Parameters.xPhysicalTempFeedback)
				THEN
				ReadingUvOnTimeStep := READINGUVTIME_INIT;
			END_IF

		READINGUVTIME_INIT:
			dataLed.Comms.Command.Close := TRUE;
			dataLed.Comms.Device.receive_data := '';

			ReadingUvOnTimeStep := READINGUVTIME_READING;

		READINGUVTIME_READING:

			ReadLampUvOnTime;
			StAnswer := MID(dataLed.Comms.Device.receive_data, iAnswerStringLength, iAnswerStringPosition);
			IF (StAnswer<>'') THEN
				ReadingUvOnTimeStep := READINGUVTIME_READY;

			ELSIF (dataLed.Comms.Device.step = FRM_WAIT)THEN
				//To send command to lamp
				dataLed.Comms.Command.Send := TRUE;
			END_IF

		READINGUVTIME_READY:

			dataLed.Lamp[iIndexReadUvOnTimeLamps].Status.rUvOnTime := brsatof(ADR(StAnswer));
			dataLed.Lamp[iIndexReadUvOnTimeLamps].Status.stUvOnTimeRaw := StAnswer;
			ReadNextLampUvOnTime;

	END_CASE

	dataLed.Comms.Device.send_data := StMessage;

END_ACTION

//Telegrams to be sent to curing led devices//
//To read lamp's intensity setpoint
ACTION ReadLampUvOnTime:
	//To define the string to be sent to the lamp
	StMessage := StCmdRead;
	//strcat: Used to link (concat) several strings
	strcat(ADR(StMessage), ADR(dataLed.Lamp[iIndexReadUvOnTimeLamps].Status.stSerialNumber));
	strcat(ADR(StMessage), ADR(StMl));
	strcat(ADR(StMessage), ADR(' uvt'));

	iAnswerStringLength := 10;
	iAnswerStringPosition := 1;

END_ACTION

ACTION ReadNextLampUvOnTime:

	//Erasing buffer and going to next lamp
	iIndexReadUvOnTimeLamps := iIndexReadUvOnTimeLamps + 1;
	IF iIndexReadUvOnTimeLamps <= iLampsQuantity THEN
		ReadingUvOnTimeStep := READINGUVTIME_INIT;
	ELSE
		ReadingUvOnTimeStep := READINGUVTIME_NOT_INIT;
	END_IF

END_ACTION
```

#### EventLog.st
```iecst
ACTION LogStopAlarm:

	stEventLog.Source := ELOG_TYPE_LED;
	stEventLog.Severity:= ELOG_SEVERITY_INFO;
	stEventLog.Facility:= iIndexCuringLed;
	stEventLog.ErrorCode:=0;

	stEventLog.Text := 'dataLed.StopAlarm';

	IF 		iReasonStop.0 THEN stEventLog.Text := 'dataLed.Alarms.xN2LowFlow';
	ELSIF 	iReasonStop.1 THEN stEventLog.Text := 'dataLed.Alarms.xLampsSlmNotConfigured';
	ELSIF 	iReasonStop.2 THEN stEventLog.Text := 'dataLed.Alarms.xFrontDoorOpened';
	END_IF

	gEventLogLoader(EventData := ADR(stEventLog));

END_ACTION

ACTION LogCriticalAlarm:

	stEventLogCritical.Source := ELOG_TYPE_LED;
	stEventLogCritical.Severity:= ELOG_SEVERITY_ERROR;
	stEventLogCritical.Facility:= iIndexCuringLed;
	stEventLogCritical.ErrorCode:=0;

	stEventLogCritical.Text := 'dataLed.CriticalAlarm';

	IF 		iReasonCritical.0 THEN stEventLogCritical.Text := 'dataLed.Alarms.xCureSystemFaulted';
	ELSIF 	iReasonCritical.1 THEN stEventLogCritical.Text := 'errorLampsSLM>0';
	ELSIF 	iReasonCritical.2 THEN stEventLogCritical.Text := 'errorLampsThermal>0';
	ELSIF	iReasonCritical.3 THEN stEventLogCritical.Text := 'dataLed.Alarms.xSerialNumbersNotAssigned';
	ELSIF	iReasonCritical.4 THEN stEventLogCritical.Text := 'dataLed.Alarms.xDetectionProcessFailed';
	ELSIF	iReasonCritical.5 THEN stEventLogCritical.Text := 'dataLed.Alarms.xPowerFailure';
	END_IF

	gEventLogLoader(EventData := ADR(stEventLogCritical));

END_ACTION

ACTION LogPsuFailure:

	stEventLogPsuFailure.Source := ELOG_TYPE_LED;
	stEventLogPsuFailure.Severity:= ELOG_SEVERITY_ERROR;
	stEventLogPsuFailure.Facility:= iIndexPowerSupply;
	stEventLogPsuFailure.ErrorCode:=0;

	stEventLogPsuFailure.Text := 'dataLed.PsuFailure. PSU:';
	brsitoa(iIndexPowerSupply, ADR(strAuxEventDesc));
	brsstrcat(ADR(stEventLogPsuFailure.Text), ADR(strAuxEventDesc));

	gEventLogLoader(EventData := ADR(stEventLogPsuFailure));

END_ACTION
```

#### CuringLedCtrl.var - Local variables
```iecst
VAR
	xDetectionLampsProcessOn : BOOL;
	xPowerOnLamps : BOOL;
	tonRunChiller : TON;
	rCureBySpeedIntercept : REAL;
	rCureBySpeedSlope : REAL;
	tonLampsVoltageRecovery : TON;
	tonFinishPolling : TON;
	xRepeated : BOOL;
	StAnswerAux : STRING[800];
	StAnswer : STRING[800];
	StMessage : STRING[80];
	StGoodAnswer : STRING[800];
	iAnswerStringPosition : INT;
	StIndex : STRING[2];
	BufferRecieve : STRING[255];
	rLastCuringBarSlmL2 : REAL; (*Fist slm to be enabled in the bar for L2*)
	iNumLampSLM : UINT;
	iMinBufferLength : UINT; (*iMinBufferLength to consider valid message from lamp*)
	CommsCommandsReset : Comms_command_typ;
	AutoIntensitySetPoint : USINT;
	rInteger : REAL; (*Integer part, result of a divsion*)
	xConfigurationFailed : BOOL;
	rMantissa : REAL; (*Decimal part, result of a division*)
	pInteger : UDINT; (*Integer part, result of a divsion*)
	rFirstCuringBarSlmL2 : REAL; (*Fist slm to be enabled in the bar for L1*)
	iFirstLampSLM : INT;
	iLastLampSLM : INT;
	iMirrorSlm : INT;
	xSendingBuffer : BOOL;
	rLastCuringBarSlmL1 : REAL; (*Fist slm to be enabled in the bar for L2*)
	rFirstCuringBarSlmL1 : REAL; (*Fist slm to be enabled in the bar for L1*)
	iLastCuringBarSlmL2 : UINT; (*Last slm to be enabled in the bar for L2*)
	iLastCuringBarSlmL1 : UINT; (*Fist slm to be enabled in the bar for L2*)
	iFirstCuringBarSlmL2 : UINT; (*Last slm to be enabled in the bar for L1*)
	iFirstCuringBarSlmL1 : UINT; (*Fist slm to be enabled in the bar for L1*)
	iTotalNumSlms : UINT; (*Number of slm in all the bar. Sum of lamps SLMs*)
	xCuringLedSlms : ARRAY[0..100] OF BOOL; (*1 Slm = 25mm. Maximum Curing led width would be 2500mm*)
	xBoardPositionChanged : BOOL;
	iPreviousWidth : UINT;
	iPreviousOffsetRegisterL2 : INT;
	iPreviousOffsetRegisterL1 : INT;
	xBufferSent : BOOL;
	xCommsClosed : BOOL;
	xBufferReadInvalid : BOOL;
	xReleasingReadBuffer : BOOL;
	xBufferReadReleased : BOOL;
	xReleasingSendBuffer : BOOL;
	xBufferSendReleased : BOOL;
	ars_AlrWarning : AutoResetSound;
	ars_AlrStop : AutoResetSound;
	ars_AlrCritical : AutoResetSound;
	xClosingComms : BOOL;
	xCommsOpened : BOOL;
	xClearingBuffer : BOOL;
	xBufferCleared : BOOL;
	xOpeningComms : BOOL;
	aPreSerialNumbers : ARRAY[1..15] OF STRING[6]; (*Index for running the elements*)
	iIndexPreSerialNumbers : UINT; (*Index for running the elements*)
	iDetectedLamp : UINT; (*Index for running the elements*)
	i : INT;
	iIndexReadUvOnTimeLamps : UINT; (*Index for running the elements*)
	iIndexReadTempLamps : UINT; (*Index for running the elements*)
	iIndexDetectLamps : UINT; (*Index for running the elements*)
	iIndexCheckSlm : UINT; (*Index for running the elements*)
	iIndexCheckLamps : UINT; (*Index for running the elements*)
	iIndexConfigSlm : UINT; (*Index for running the elements*)
	iIndexEraseReceivedData : UINT; (*Index for running the elements*)
	iIndexConfigLamps : UINT; (*Index for running the elements*)
	iIndexEnableLamps : UINT; (*Index for running the elements*)
	iIndexEnableSlm : UINT; (*Index for running the elements*)
	xCuringOrder : BOOL; (*General curing order while everything is ready*)
	tonNitroAlrLowFlow : TON;
	iLampPosition : INT;
	iPowerSuppliesQuantity : INT;
	iLampsQuantity : UINT;
	errorLampsSLM : UDINT;
	errorLampsThermal : UDINT;
	iBoardFinalPosition : INT;
	iBoardInitPosition : INT;
	xAnyError : BOOL;
	xEnableCuring : BOOL;
	xBufferRead : BOOL;
	arxLampsSlmNotConfigured : AutoResetSound;
	arxPowerFailure : AutoResetSound;
	arxCureSystemFaulted : AutoResetSound;
	xReadBufferNoInput : BOOL;
	arxN2HighFlow : AutoResetSound;
	StatusCtrl : CuringLedStatus_enum;
	ConfigCtrl : CuringLedConfig_enum;
	CheckStep : CuringLedCheck_enum;
	DetectStep : CuringLedDetect_enum;
	ReadingUvOnTimeStep : CuringLedReadingLampUvTime_enum;
	ReadingTemperatureStep : CuringLedReadingLampTemp_enum;
	iIndexPowerSupply : INT; (*Index for running the elements*)
	iIndexCuringAux : UINT; (*Index for running the elements*)
	iIndexCuring : UINT; (*Index for running the elements*)
	arLampThermalFault : AutoResetSound;
	arLampSLMFault : AutoResetSound;
	xReadBufferInputError : BOOL;
	iReasonCritical : UDINT;
	NitroState : CuringLed_NitrogenStatus_enum;
	iReasonWarning : UDINT;
	iReasonStop : UDINT;
	stEventLog : EventLog_typ;
	stEventLogCritical : EventLog_typ;
	stEventLogPsuFailure : EventLog_typ;
	strAuxEventDesc : STRING[129];
	AlarmsReseted : CuringLed_Alarms_typ;
	AlarmsSummaryReseted : stEFI_AlarmSummary;
	dataChiller : REFERENCE TO StChiller;
	dataLed : REFERENCE TO CuringLed_typ;
	send_data : STRING[800];
	FindInString : STRING[10];
	xValidStatusReading : BOOL;
	StSupplySide : STRING[8];
	iSupplySide : UINT;
	arxChillerFaulted : AutoResetSound;
	xSLMStatusRead : BOOL;
	iAnswerStringLength : INT;
	xKeepFilling : BOOL;
	iCheckStatusAttempts : INT;
	iDetectLampAttempts : INT;
	OutputsReset : CuringLed_Signals_Out_typ;
	ResetCommands : CuringLed_Commands_typ;
	iIndexPreSerialNum : UINT;
	xFinishPolling : BOOL;
	ResetManCommands : CuringLed_ManualCommands_typ;
	iIntensityCureBySpeed : USINT; (*//Setpoint to be used while curing by speed is active*)
	iIntensityWhileAtSafePosition : USINT := 30; (*//Setpoint to be used while emptying belt to cure media but not cure bar's nozzles*)
	iMinSpeedWhenBlockAtSafePosition : REAL := 50; (*//Belt speed setpoint from which intensity applied while block is at safe position changes*)
	StateHistory : ARRAY[0..iHistoryLines] OF enComms_STEPS;
END_VAR
VAR CONSTANT
	iHistoryLines : USINT := 20;
END_VAR
VAR
	iIndexHistory : USINT;
	tonOpenPort : TON;
	tonPowerOnLamps : TON;
	xAnyErrorReason : UINT;
	xAnyParamChanged : UINT;
	iTotalWidth : INT; (*Sum of curing led bar lamp's widths*)
	iCenterPosition : INT; (*Curing led bar center position*)
	tonCheckAlarms : TON;
	tonStabPsuFailure : ARRAY[0..10] OF TON;
END_VAR
```

- CuringLed.graphml (not shown)

### Program Logical/ExtPack/_Cure/CuringLedCtrl/CuringLedSim/CuringLedSim_v1/CuringLedSim (IEC)

#### CuringLedSim.var
```iecst
VAR
	dataLed : REFERENCE TO CuringLed_typ;
END_VAR
```

### Program Logical/ExtPack/_Cure/CuringLedCtrl/CuringLedSim/CuringLedSim_v1/InitCuringLedSim (IEC)

#### InitCuringLedSim.st
```iecst
PROGRAM _CYCLIC
	iIndexCuringLedSim := 1;
END_PROGRAM
```

### CuringLedSim.var - Local variables
```iecst
VAR
	iIndexCuringLedSim : USINT;
END_VAR
```

### NIRAdphosCtrl.typ
```iecst
TYPE
	NIRAdphos_State :
		(
		NIRADPEW_NOT_INITIALIZED,
		NIRADPEW_INIT,
		NIRADPEW_IDLE,
		NIRADPEW_POWER_ON,
		NIRADPEW_POWERED,
		NIRADPEW_RUNNING_BELT,
		NIRADPEW_READY,
		NIRADPEW_STARTING,
		NIRADPEW_RUNNING,
		NIRADPEW_ERROR,
		NIRADPEW_SAFETY_ERROR,
		NIRADPEW_COMMS_ERROR
		);
	NIRAdphos_ModuleState :
		(
		NIRADPM_UNDEFINED, (*Wrong value*)
		NIRADPM_OFF, (*0*)
		NIRADPM_STARTUP, (*1*)
		NIRADPM_READY, (*2*)
		NIRADPM_STANDBY, (*3*)
		NIRADPM_PROCESS, (*4*)
		NIRADPM_SHUTDOWN (*5*)
		);
	NIRAdphos_CommsInModule : 	STRUCT  (*From Dryer to Adphos*)
		NirStatus : NIRAdphos_ModuleState := NIRADPM_UNDEFINED; (*Value transformed from iNirStatus, directly received from comms*)
		iNirStatus : INT; (*NIR Status: 0=Off, 1=StartUp, 2=Ready, 3=StandBy, 4=Process, 5=Shutdown*)
		Watchdog : BOOL; (*1Hz blink with communication*)
		error : BOOL;
		message : BOOL; (*There is at least one message*)
		closed : BOOL; (*Module closed in docking station*)
		SuppAirRunning : BOOL; (*Support air blower running*)
		ExtAirRunning : BOOL; (*Exhaust air blower running*)
		TotalInFail : USINT; (*EmFailNo. Number of emmiters with defect*)
		AirPressIn : REAL; (*Aire pressure support air [Pa]*)
		AirPressOut : REAL; (*Aire pressure exhaust air [Pa]*)
		AirFilter : INT; (*Aire pressure Filter monitoring [Pa]*)
		SpeedIn : INT; (*Speed In [%]*)
		SpeedOut : INT; (*Speed Out [%]*)
		xPowered : BOOL; (*Calculated from other info received*)
		Power : INT; (*Power [%]*)
	END_STRUCT;
	NIRAdphos_CommsInVersion : 	STRUCT  (*From Dryer to Adphos*)
		Software : INT; (*Software version*)
		Hardware : INT; (*Hardware version*)
		Interface : INT; (*Interface version*)
		HMI : INT; (*HMI version*)
	END_STRUCT;
	NIRAdphos_CommsInCalc_Spare : 	STRUCT
		xPowered : BOOL; (*Calculated from other info received*)
		xBeltRunning : BOOL; (*Calculated from other info received*)
	END_STRUCT;
	NIRAdphos_CommsIn : 	STRUCT  (*From Adphos to Dryer*)
		Version : NIRAdphos_CommsInVersion;
		Speed : REAL; (*Current speed [m/min]*)
		CalPower : INT; (*Calculated power [%]*)
		NirWidth : INT; (*Current NIR Width [mm]*)
		NirTotalActive : INT; (*Number of active emiters*)
		xBeltRunning : BOOL; (*Calculated from other info received*)
		Modules : ARRAY[0..2]OF NIRAdphos_CommsInModule; (*Module 0 not used*)
		Zones : ARRAY[0..48]OF BOOL; (*Current active zones. Zone 0 not used*)
	END_STRUCT;
	NIRAdphos_CommsOutModule : 	STRUCT  (*From Dryer to Adphos*)
		Adjust : INT; (*Adjust heatihng power [0 to 100 %]*)
		EnableMod : BOOL; (*Enable module*)
	END_STRUCT;
	NIRAdphos_CommsOut : 	STRUCT  (*From Dryer to Adphos*)
		Vstart : REAL; (*Start speed [m/min]*)
		Vend : REAL; (*Final speed [m/min]*)
		Pstart : REAL; (*Start Power [%]*)
		Pend : REAL; (*Final Power [%]*)
		WebWidth : INT; (*WebWidth [360 to 1440mm]. DO NOT WRITE DIRECTLY FROM OUTSIDE NIR CODE*)
		AdjPos : INT; (*Adjust heatihng area [+ or - xx mm]*)
		Modules : ARRAY[0..2]OF NIRAdphos_CommsOutModule; (*Module 0 not used*)
	END_STRUCT;
	NIRAdphos_Comms : 	STRUCT  (*DEPRECATED. USED INSIDE STRUCTURE IN PARAMS AND STATUS*)
		In : NIRAdphos_CommsIn; (*From Adphos to Dryer*)
		Out : NIRAdphos_CommsOut; (*From Dryer to Adphos*)
	END_STRUCT;
	NIRAdphos_DDC : 	STRUCT  (*DEPRECATED. USED INSIDE STRUCTURE IN PARAMS AND STATUS*)
		xEnableDDC : BOOL; (*Enable Dynamic Dryer Control *)
		iLamps : USINT; (*Total quantity of Lamps in the machine*)
		iLampsExtend : USINT := 0; (*Quantity of lamps to extend the value of each lamp*)
		rMinIntensityPercentage : REAL; (*Minimum value of Drying during DDC. With the speed and the curve, the value to send to the Dryer is modifyed and increased if needed. 10 expected for 10%*)
		pIntensityNir1 : {REDUND_UNREPLICABLE} UDINT;
		pIntensityNir2 : {REDUND_UNREPLICABLE} UDINT;
	END_STRUCT;
	NIRAdphos_Parameters : 	STRUCT
		StateMode : enumEFI_GenMachineState; (*commands to block*)
		AutoMode : stEFI_MachineAutoModes;
		xEnableNir : BOOL;
		DDC : NIRAdphos_DDC;
		CpuFamily : USINT;
		rBeltSpeed : REAL; (*Current speed of the belt*)
		xBeltRunning : BOOL; (*External information about the belt moving*)
		rMaxSurfaceTemp : REAL; (*Maximum allowed surface temperature*)
		iTotalModules : USINT; (*Total NIR modules*)
		Comms : NIRAdphos_CommsOut;
		xLineEmptyingBelt : BOOL; (*Line in empty belt mode*)
		MediaWidth : INT; (*MediaWidth. WebWidth [360 to 1440mm]*)
		iExtraDryingWidh : INT := 0; (*Extra drying width in mm. Value added to allow more lamps turnend on than the theoretical. Just positive values*)
		xInstalled : BOOL;
	END_STRUCT;
	NIRAdphos_AlarmsJam : 	STRUCT
		xFront : BOOL; (*Detection with first corner Front*)
		xRear : BOOL; (*Detection with first corner Rear*)
		xCross : BOOL; (*Detecction across NIR*)
		xMechCross : BOOL; (*Mechanical detectin across NIR*)
	END_STRUCT;
	NIRAdphos_AlarmsBlockedFans : 	STRUCT  (*EFI Signal*)
		Fan : ARRAY[0..4]OF BOOL; (*0 not used*)
	END_STRUCT;
	NIRAdphos_Alarms : 	STRUCT
		xCommsError : BOOL; (*EDGE*)
		xMaxSurfaceTempModule : ARRAY[0..MAX_LAST_NIR_MODULES]OF BOOL; (*Max Surface temperature achieved. 0 is not used*)
		xSurfaceTempModuleSensorError : ARRAY[0..MAX_LAST_NIR_MODULES]OF BOOL; (*Sensor error. 0 is not used*)
		BlockedFansModule : ARRAY[0..MAX_LAST_NIR_MODULES]OF NIRAdphos_AlarmsBlockedFans;
		Jam : ARRAY[0..MAX_LAST_NIR_MODULES]OF NIRAdphos_AlarmsJam;
		xOpcUaWriteError : ARRAY[0..MAX_LAST_NIR_MODULES]OF BOOL; (*Comms error in the OpcUa Write comms*)
		xAnyJam : BOOL; (*Summary signal of any of the jams in the modules*)
		xSafetyError : BOOL; (*Safety error in the Dryer*)
		xFault : BOOL; (*Fault detected in the Dryer*)
		xInletTempSensorError : BOOL; (*EFI signal from Inlet Temperature. Sensor Error*)
		xInletHumiditySensorError : BOOL; (*EFI signal from Inlet Humidity. Sensor Error*)
	END_STRUCT;
	NIRAdphos_CommandsComms : 	STRUCT
		xSpare : BOOL;
	END_STRUCT;
	NIRAdphos_Commands : 	STRUCT
		xPrepare : BOOL; (*EDGE*)
		xStart : BOOL; (*EDGE*)
		xStop : BOOL; (*EDGE*)
		xReset : BOOL;
		xMute : BOOL;
		xMediaInside : BOOL;
		xExternalSafetyStop : BOOL; (*External Safety Stop order*)
		Comms : NIRAdphos_CommandsComms;
	END_STRUCT;
	NIRAdphos_JamInputs : 	STRUCT
		xMechCross : BOOL; (*Mechanical detectin across NIR*)
	END_STRUCT;
	NIRAdphos_BlockedFansSignalsIn : 	STRUCT  (*EFI Signal*)
		Fan : ARRAY[0..4]OF BOOL; (*0 not used. 1 Is the first in the operator side*)
	END_STRUCT;
	NIRAdphos_SignalsIn : 	STRUCT
		xReady : BOOL;
		xFault : BOOL; (*Any error in the enabled alarms*)
		xInProcess : BOOL;
		xSafetyOK : BOOL; (*Safety in the NIR Dryer is OK*)
		iInletTempRaw : INT; (*EFI signal from Inlet Temperature*)
		iInletHumidityRaw : INT; (*EFI signal from Inlet Humidity*)
		xInletTempSensorError : BOOL; (*EFI signal from Inlet Temperature. Sensor Error*)
		xInletHumiditySensorError : BOOL; (*EFI signal from Inlet Humidity. Sensor Error*)
		iSurfaceTempModuleRaw : ARRAY[0..MAX_LAST_NIR_MODULES]OF INT; (*EFI signal from Surface Temperature of the modules directly from the Input Card. 0 is not used*)
		xSurfaceTempModuleSensorError : ARRAY[0..MAX_LAST_NIR_MODULES]OF BOOL; (*EFI signal from Surface Temperature of the modules directly from the Input Card. 0 is not used*)
		Jam : ARRAY[0..MAX_LAST_NIR_MODULES]OF NIRAdphos_JamInputs; (*EFI signal from Surface Temperature of the modules directly from the Input Card. 0 is not used*)
		BlockedFans : ARRAY[0..MAX_LAST_NIR_MODULES]OF NIRAdphos_BlockedFansSignalsIn; (*EFI signal. 0 not used*)
	END_STRUCT;
	NIRAdphos_SignalsOut : 	STRUCT
		xPowerOn : BOOL;
		xProcess : BOOL;
		xSafetyStop : BOOL; (*Any error in the enabled alarms*)
		iBeltSpeed : INT; (*Current speed of the belt*)
		xWatchDog : BOOL; (*1Hz blinking data*)
	END_STRUCT;
	NIRAdphos_Signals : 	STRUCT
		In : NIRAdphos_SignalsIn;
		Out : NIRAdphos_SignalsOut; (*Any error in the enabled alarms*)
	END_STRUCT;
	NIRAdphos_DDCIntensityStatus : 	STRUCT
		Intensity : ARRAY[0..THICKENERGY_MAX_LAMPS]OF INT; (*Data starting in index 1*)
	END_STRUCT;
	NIRAdphos_Status : 	STRUCT
		xAnyModuleEnabled : BOOL;
		xAnyModuleInError : BOOL; (*Any error in the enabled alarms*)
		xEnabledNir : BOOL;
		xEnabledDDC : BOOL;
		DDC : ARRAY[0..MAX_LAST_NIR_MODULES]OF NIRAdphos_DDCIntensityStatus;
		rPowerSetPoint : REAL; (*Power SetPoint calculated from Speed and Power/Speed curve*)
		iMinPower : INT; (*Minimum power calculated with the curves and the spped*)
		rInletTemperature : REAL;
		rInletHumidity : REAL;
		rSurfaceTempModule : ARRAY[0..MAX_LAST_NIR_MODULES]OF REAL; (*Surface Temperature of the modules in degree Celsius. 0 is not used*)
		xDrying : BOOL; (*Summary information. State == RUNNING*)
		xCommsOK : BOOL;
		Comms : NIRAdphos_CommsIn;
	END_STRUCT;
	NIRAdphos_Orders : 	STRUCT
		xCheckJam : BOOL; (*Order active when dryer conditions require to check jam sensors*)
	END_STRUCT;
	NIRAdphos : 	STRUCT
		Parameters : NIRAdphos_Parameters;
		State : NIRAdphos_State := NIRADPEW_NOT_INITIALIZED;
		Alarms : NIRAdphos_Alarms;
		AlSummary : stEFI_AlarmSummary;
		Commands : NIRAdphos_Commands;
		Signals : NIRAdphos_Signals;
		Status : NIRAdphos_Status;
		Orders : NIRAdphos_Orders;
	END_STRUCT;
END_TYPE
```

### Library Logical/ExtPack/_Cure/NIRAdphos/NIRAdphos_v1/NIRAdphosCtrl

#### CommsNir1.var
```iecst
VAR CONSTANT
	iIndexConstant_Nir1 : USINT := 1;
END_VAR
VAR
	ExecuteConnect_Nir1 : BOOL;
	SessionConnectInfo_Nir1 : UASessionConnectInfo;
	ConnectionHdl_Nir1 : DWORD;
	UA_Connect_Nir1 : UA_Connect;
	ExecuteGetnamespaceindex_Nir1 : BOOL;
	NamespaceIndex_Nir1 : UINT;
	UA_GetNamespaceIndex_Nir1 : UA_GetNamespaceIndex;
	ExecuteMethodGetHandle_Nir1 : BOOL;
	ObjectNodeID_Nir1 : UANodeID;
	NodeHdl_Nir1 : DWORD;
	NodeAddInfo_Nir1 : UANodeAdditionalInfo;
	IndexRange_Nir1 : UAIndexRange;
	InputArguments_Nir1 : ARRAY[0..9] OF UAMethodArgument;
	OutputArguments_Nir1 : ARRAY[0..9] OF UAMethodArgument;
	UA_NodeGetHandle_Nir1 : UA_NodeGetHandle;
	ExecuteMethodCall_Nir1 : BOOL;
	UA_Write_Nir1 : UA_Write;
	MethodResult_Nir1 : UDINT;
	NewMediaData_Nir1 : stThicknessCtrl_MediaConfig;
	tonNotCallingMethod_Nir1 : TON;
	UA_NodeReleaseHandle_Nir1 : UA_NodeReleaseHandle;
	ExecuteNodeReleaseHandle_Nir1 : BOOL;
	UA_Disconnect_Nir1 : UA_Disconnect;
	ExecuteDisconnect_Nir1 : BOOL;
	iValues_Nir1 : ARRAY[0..47] OF INT; (*Data starting in index 0*)
	iTimes_Nir1 : UDINT;
	CommsState_Nir1 : OpcUaCommsState;
	iIndexValue_Nir1 : USINT;
	tonNextComms_Nir1 : TON;
	iGoodComms_Nir1 : UINT;
	tonCalculateUpdate_Nir1 : TON;
	iPartialGoodTimes_Nir1 : UINT;
	rUpdateRatio_Nir1 : REAL; (*milliseconds per update*)
	tonWaitExitFault_Nir1 : TON;
	xAnyCommsError_Nir1 : BOOL;
	StateHistory_Nir1 : ARRAY[0..iHistoryLines] OF OpcUaCommsState;
	iIndex_Nir1 : USINT;
	Intensity_Nir1 : REFERENCE TO ARRAY[0..THICKENERGY_MAX_LAMPS] OF INT; (*Data starting in index 1*)
	IntensityExtend_Nir1 : {REDUND_UNREPLICABLE} ARRAY[0..THICKENERGY_MAX_LAMPS] OF INT; (*Data starting in index 1*)
	IntensityReseted_Nir1 : {REDUND_UNREPLICABLE} ARRAY[0..THICKENERGY_MAX_LAMPS] OF INT;
	iIndexExtend_Nir1 : USINT;
END_VAR
```

#### CommsNir2.var
```iecst
VAR CONSTANT
	iIndexConstant_Nir2 : USINT := 2;
END_VAR
VAR
	ExecuteConnect_Nir2 : BOOL;
	SessionConnectInfo_Nir2 : UASessionConnectInfo;
	ConnectionHdl_Nir2 : DWORD;
	UA_Connect_Nir2 : UA_Connect;
	ExecuteGetnamespaceindex_Nir2 : BOOL;
	NamespaceIndex_Nir2 : UINT;
	UA_GetNamespaceIndex_Nir2 : UA_GetNamespaceIndex;
	ExecuteMethodGetHandle_Nir2 : BOOL;
	ObjectNodeID_Nir2 : UANodeID;
	NodeHdl_Nir2 : DWORD;
	NodeAddInfo_Nir2 : UANodeAdditionalInfo;
	IndexRange_Nir2 : UAIndexRange;
	InputArguments_Nir2 : ARRAY[0..9] OF UAMethodArgument;
	OutputArguments_Nir2 : ARRAY[0..9] OF UAMethodArgument;
	UA_NodeGetHandle_Nir2 : UA_NodeGetHandle;
	ExecuteMethodCall_Nir2 : BOOL;
	UA_Write_Nir2 : UA_Write;
	MethodResult_Nir2 : UDINT;
	NewMediaData_Nir2 : stThicknessCtrl_MediaConfig;
	tonNotCallingMethod_Nir2 : TON;
	UA_NodeReleaseHandle_Nir2 : UA_NodeReleaseHandle;
	ExecuteNodeReleaseHandle_Nir2 : BOOL;
	UA_Disconnect_Nir2 : UA_Disconnect;
	ExecuteDisconnect_Nir2 : BOOL;
	iValues_Nir2 : ARRAY[0..47] OF INT; (*Data starting in index 0*)
	iTimes_Nir2 : UDINT;
	CommsState_Nir2 : OpcUaCommsState;
	iIndexValue_Nir2 : USINT;
	tonNextComms_Nir2 : TON;
	iGoodComms_Nir2 : UINT;
	tonCalculateUpdate_Nir2 : TON;
	iPartialGoodTimes_Nir2 : UINT;
	rUpdateRatio_Nir2 : REAL; (*milliseconds per update*)
	tonWaitExitFault_Nir2 : TON;
	xAnyCommsError_Nir2 : BOOL;
	StateHistory_Nir2 : ARRAY[0..iHistoryLines] OF OpcUaCommsState;
	iIndex_Nir2 : USINT;
	Intensity_Nir2 : REFERENCE TO ARRAY[0..THICKENERGY_MAX_LAMPS] OF INT;
	IntensityExtend_Nir2 : {REDUND_UNREPLICABLE} ARRAY[0..THICKENERGY_MAX_LAMPS] OF INT; (*Data starting in index 1*)
	IntensityReseted_Nir2 : {REDUND_UNREPLICABLE} ARRAY[0..THICKENERGY_MAX_LAMPS] OF INT;
	iIndexExtend_Nir2 : USINT;
END_VAR
```
